// TIA Portal project "Blending_Process" (V16)

(* hardware
DEVICE "S7-1200 station_1"  S7-1200 Station
   slot 0: "Rack_0"  S7-1200 Rack  Rack  V1.0
   slot 1: "PLC_1"  CPU 1214C DC/DC/DC  6ES7 214-1AG40-0XB0  V4.2
DEVICE "HMI_1"  KTP700 Basic PN
   slot 0: "HMI_1"  KTP700 Basic PN  6AV2 123-2GB03-0AX0  16.0.0.0
   slot 1: "HMI_RT_1"  KTP700 Basic PN  6AV2 123-2GB03-0AX0  16.0.0.0
   slot 5: "HMI_1.IE_CP_1"  PROFINET Interface  16.0.0.0
      slot 1: "PROFINET Interface_1"  PROFINET Interface
         slot 1: "Port_1"  Port
*)

// ===== PLC "PLC_1"  CPU 1214C DC/DC/DC =====

VAR_GLOBAL   // PLC tag table "Default tag table"
   "Tag_1" AT %M2.0 : Bool;
   "Tag_2" AT %M2.1 : Bool;
   "RESET_FAULT" AT %M3.3 : Bool;
   "Tag_3" AT %M3.4 : Bool;
   "Reset_Fault_2" AT %M3.5 : Bool;
   "RSET_FAULT_DRAIN" AT %M3.6 : Bool;
   "iq_rMotor_Speed" AT %MD1 : Real;
   "i_xMix_Motor_Stop" AT %I4.0 : Bool;
   "q_xMix_Motor_Stop" AT %Q6.5 : Bool;
   "Tag_4" AT %M50.1 : Bool;
   "Tag_5" AT %M100.0 : Bool;
   "Tag_6" AT %M101.0 : Bool;
   "Tag_7" AT %M102.0 : Bool;
   "Tag_8" AT %M103.0 : Bool;
   "Tag_9" AT %M104.0 : Bool;
   "Tag_10" AT %M110.0 : Bool;
   "Tag_11" AT %M113.0 : Bool;
   "Tag_12" AT %M115.0 : Bool;
   "_iCount_Motor" AT %MW130 : Int;
   "_iCount_Pump1" AT %MW115 : Int;
   "_iCount_Pump2" AT %MW118 : Int;
   "Drain" AT %M74.0 : Bool;
   "Tag_13" AT %M120.0 : Bool;
END_VAR

VAR_GLOBAL   // PLC tag table "Inputs Equipment"
   "i_xSupply_InletValve_Open_A1" AT %I0.1 : Bool;
   "i_xSupply_FeedPump_Running_A1" AT %I2.1 : Bool;
   "i_xSupply_FeedValve_Open_A1" AT %I0.0 : Bool;
   "i_xSupply_FlowSensor_A1" AT %I0.5 : Bool;
   "i_xMix_Motor_Running" AT %I4.1 : Bool;
   "i_xDrain_SolenoidValve_Open" AT %I2.5 : Bool;
   "i_xSupply_InletValve_Open_A2" AT %I0.3 : Bool;
   "i_xSupply_FeedPump_Running_A2" AT %I2.7 : Bool;
   "i_xSupply_FeedValve_Open_A2" AT %I0.2 : Bool;
   "i_xSupply_FlowSensor_A2" AT %I0.6 : Bool;
   "i_xMix_Tank_EmptySensor" AT %I0.4 : Bool;
   "i_rMix_Motor_Voltage" AT %MD10 : Real;
   "i_rMix_Tank_Level" AT %MD64 : Real;
   "i_xSupply_FeedPump_Ready_A1" AT %I3.5 : Bool;
   "i_xSupply_FeedPump_Ready_A2" AT %I3.6 : Bool;
   "i_xDrain_SolenoidValve_Close" AT %I2.3 : Bool;
END_VAR

VAR_GLOBAL   // PLC tag table "Outputs Equipment"
   "q_xSupply_FeedPump_Start_A1" AT %Q3.0 : Bool;
   "q_xMix_Motor_Start" AT %Q6.4 : Bool;
   "q_xDrain_SolenoidValve_Open" AT %Q3.7 : Bool;
   "q_xSupply_FeedPump_Start_A2" AT %Q3.1 : Bool;
   "q_xSupply_InletValve_Open_A2" AT %Q3.3 : Bool;
   "q_xSupply_FeedValve_Open_A2" AT %Q3.5 : Bool;
   "q_xSupply_FeedPump_Stop_A1" AT %Q6.0 : Bool;
   "q_xSupply_FeedPump_Stop_A2" AT %Q6.1 : Bool;
   "q_xDrain_SolenoidValve_Close" AT %Q2.7 : Bool;
   "q_xSupply_FeedValve_Open_A1" AT %Q3.4 : Bool;
   "q_xSupply_InletValve_Open_A1" AT %Q3.2 : Bool;
   "iq_xMix_Tank_FullSensor" AT %I7.7 : Bool;
   "iq_rWater_Level" AT %MD7 : Real;
END_VAR

VAR_GLOBAL   // PLC tag table "Inputs Machine"
   "i_xButtonFeedPump_Start_A1" AT %I30.3 : Bool;
   "i_xButtonFeedPump_Stop_A1" AT %I30.4 : Bool;
   "i_xButtonMotor_Start" AT %I30.0 : Bool;
   "i_xButtonMotor_Stop" AT %I30.1 : Bool;
   "i_xButtonSolenoidValve_Start" AT %I31.0 : Bool;
   "i_xButtonSolenoidValve_Stop" AT %I31.1 : Bool;
   "i_xButtonMaintenanceLamp_Stop" AT %I10.6 : Bool;
   "i_xButton_Emergency" AT %I10.7 : Bool;
   "i_xButtonFeedPump_Start_A2" AT %I30.5 : Bool;
   "i_xButtonFeedPump_Stop_A2" AT %I30.6 : Bool;
   "i_xButton_Reset" AT %I30.2 : Bool;
   "i_xButton_Turn/off_Maintenance_Pump" AT %I31.3 : Bool;
   "i_xButton_Turn/off_Maintenance_Motor" AT %I31.2 : Bool;
   "i_xFull_Sensor" AT %I8.0 : Bool;
END_VAR

VAR_GLOBAL   // PLC tag table "Outputs Machine"
   "q_xLamp_Running" AT %Q4.0 : Bool;
   "q_xLamp_Faulted" AT %Q4.1 : Bool;
   "q_xLamp_Pump_Start_A1" AT %Q4.2 : Bool;
   "q_xLamp_Pump_Stop_A1" AT %Q4.3 : Bool;
   "q_xLamp_Pump_Start_A2" AT %Q4.4 : Bool;
   "q_xLamp_Pump_Stop_A2" AT %Q4.5 : Bool;
   "q_xLamp_Motor_Start" AT %Q4.6 : Bool;
   "q_xLampSolenoidValve_Start" AT %Q5.0 : Bool;
   "q_xLampSolenoidValve_Stop" AT %Q5.1 : Bool;
   "q_xLamp_Pump_Maintain_A1" AT %Q5.2 : Bool;
   "q_xLamp_Pump_Maintain_A2" AT %Q5.3 : Bool;
   "q_xLamp_Motor_Stop" AT %Q4.7 : Bool;
   "q_xLamp_Motor_Maintain" AT %Q5.4 : Bool;
   "q_xLamp_Tank_Full" AT %Q5.5 : Bool;
   "q_xLamp_Tank_Empty" AT %Q5.6 : Bool;
   "q_xLamp_Emergency" AT %Q5.7 : Bool;
   "q_xDisp_Tank_Level" AT %QD60 : Real;
   "q_xDisp_Motor_Speed" AT %QD64 : Real;
   "q_xMaintain_Lamp_Motor" AT %Q10.1 : Bool;
   "q_xMaintain_Lamp_Pump" AT %Q10.2 : Bool;
   "q_xLamp_Fault" AT %Q120.1 : Bool;
END_VAR

// folder: Equipment

TYPE "UDT_Supply"
   STRUCT
      Sts : Struct
         xPumpRunning : Bool;
         xPumpReady : Bool;
         xInletValveOpen : Bool;
         xFeedValveOpen : Bool;
         xFlowSensor : Bool;
         xFauted : Bool;
      END_STRUCT;
      Cmd : Struct
         xSpare : Bool;
         xStart_Pump : Bool;
         xStop_Pump : Bool;
      END_STRUCT;
      Cfg : Struct
         xSpare : Bool;
      END_STRUCT;
      Flt : Struct
         wTrigger : Word;
      END_STRUCT;
   END_STRUCT;
END_TYPE

TYPE "UDT_Mix"
   STRUCT
      Sts : Struct
         xMotorRunning : Bool;
         xMotorReady : Bool;
         iLevel : Int;
         xFullLevel : Bool;
         xEmptyLevel : Bool;
         xFaulted : Bool;
      END_STRUCT;
      Cmd : Struct
         xSpare : Bool;
         xStart_Motor : Bool;
         xStop_Motor : Bool;
      END_STRUCT;
      Cfg : Struct
         xSpare : Bool;
      END_STRUCT;
      Flt : Struct
         wTrigger : Word;
      END_STRUCT;
   END_STRUCT;
END_TYPE

TYPE "UDT_Drain"
   STRUCT
      Sts : Struct
         xSolenoidValveOpen : Bool;
         xSolenoidValveClose : Bool;
         xFaulted : Bool;
      END_STRUCT;
      Cmd : Struct
         xSpare : Bool;
         xStart_SolenoidValve : Bool;
         xStop_SsolenoidValve : Bool;
      END_STRUCT;
      Cfg : Struct
         xSpare : Bool;
      END_STRUCT;
      Flt : Struct
         wTrigger : Word;
      END_STRUCT;
   END_STRUCT;
END_TYPE

// folder: Machine

TYPE "UDT_Statehandler"
   STRUCT
      State : Struct
         xMaintenance_Pump : Bool;
         xMaintenance_Motor : Bool;
         xReady_Pump_A1 : Bool;
         xReady_Pump_A2 : Bool;
         xReady_Motor : Bool;
         xReady_SolenoidValve : Bool;
         xRunning_Pump_A1 : Bool;
         xRunning_Pump_A2 : Bool;
         xRunning_Motor : Bool;
         xRunning_SolenoidValve : Bool;
         xFaulted : Bool;
         xReset : Bool;
      END_STRUCT;
      Cmd : Struct
         xStart : Bool;
         xStop : Bool;
         xReset : Bool;
         xMaintain : Bool;
         xStart_Pump_A1 : Bool;
         xStart_Pump_A2 : Bool;
         xStart_Motor : Bool;
         xStart_SolenoidValve : Bool;
         xStop_Pump_A1 : Bool;
         xStop_Pump_A2 : Bool;
         xStop_Motor : Bool;
         xStop_Solenoid : Bool;
      END_STRUCT;
   END_STRUCT;
END_TYPE

// folder: 00 Machine

DATA_BLOCK "Instance Machine Modules_DB"   // DB3
{ S7_Optimized_Access := 'TRUE' }
VERSION : 0.1
// stored: InstanceOfName FB - Machine Modules
"FB - Machine Modules"
BEGIN
END_DATA_BLOCK

// folder: 01 Equipment

DATA_BLOCK "Instance Equipment Modules"   // DB4
{ S7_Optimized_Access := 'TRUE' }
VERSION : 0.1
// stored: InstanceOfName FB - Equipment Modules
"FB - Equipment Modules"
BEGIN
END_DATA_BLOCK

// folder: 01 Equipment/Functions

DATA_BLOCK "FB - Motor's Speed_DB"   // DB16
{ S7_Optimized_Access := 'TRUE' }
VERSION : 0.1
// stored: InstanceOfName FB - Motor's Speed
"FB - Motor's Speed"
BEGIN
   Power := 0.01;
END_DATA_BLOCK

DATA_BLOCK "FB- Water's Level_DB"   // DB17
{ S7_Optimized_Access := 'TRUE' }
VERSION : 0.1
// stored: InstanceOfName FB- Water's Level
"FB- Water's Level"
BEGIN
   i_rQ := 1.0;
   i_rK := 0.01;
   i_rA := 3.0;
   i_iT := 1;
END_DATA_BLOCK

DATA_BLOCK "FB - Agitator_DB"   // DB19
{ S7_Optimized_Access := 'TRUE' }
VERSION : 0.1
// stored: InstanceOfName FB - Agitator Motor
"FB - Agitator Motor"
BEGIN
END_DATA_BLOCK

// folder: 02 Global Data

DATA_BLOCK "DB  - Machine"   // DB1
{ S7_Optimized_Access := 'FALSE' }
VERSION : 0.1
   VAR
      StateHandler : "UDT_Statehandler";
   END_VAR
BEGIN
END_DATA_BLOCK

DATA_BLOCK "DB -  Equipment"   // DB2
{ S7_Optimized_Access := 'FALSE' }
VERSION : 0.1
   VAR
      Supply_A1 : "UDT_Supply";
      Supply_A2 : "UDT_Supply";
      Mix : "UDT_Mix";
      Drain : "UDT_Drain";
   END_VAR
BEGIN
END_DATA_BLOCK

// folder: System blocks/Program resources

DATA_BLOCK "#stOnDelay_Valve_Open"   // DB5
{ S7_Optimized_Access := 'TRUE' }
AUTHOR : Simatic
FAMILY : IEC
NAME : IEC_TMR
VERSION : 1.0
// stored: InstanceOfName IEC_TIMER
"IEC_TIMER"
BEGIN
END_DATA_BLOCK

DATA_BLOCK "#stOnDelay_Flt_Inlet Valve_2_Open"   // DB6
{ S7_Optimized_Access := 'TRUE' }
AUTHOR : Simatic
FAMILY : IEC
NAME : IEC_TMR
VERSION : 1.0
// stored: InstanceOfName IEC_TIMER
"IEC_TIMER"
BEGIN
END_DATA_BLOCK

DATA_BLOCK "#stOnDelay_Flt_FlowSensor_Report"   // DB7
{ S7_Optimized_Access := 'TRUE' }
AUTHOR : Simatic
FAMILY : IEC
NAME : IEC_TMR
VERSION : 1.0
// stored: InstanceOfName IEC_TIMER
"IEC_TIMER"
BEGIN
END_DATA_BLOCK

DATA_BLOCK "#stOnDelay_Flt_Inlet Valve_Open"   // DB8
{ S7_Optimized_Access := 'TRUE' }
AUTHOR : Simatic
FAMILY : IEC
NAME : IEC_TMR
VERSION : 1.0
// stored: InstanceOfName IEC_TIMER
"IEC_TIMER"
BEGIN
END_DATA_BLOCK

DATA_BLOCK "#stOnDelay_Flt_Feed Valve_Open"   // DB9
{ S7_Optimized_Access := 'TRUE' }
AUTHOR : Simatic
FAMILY : IEC
NAME : IEC_TMR
VERSION : 1.0
// stored: InstanceOfName IEC_TIMER
"IEC_TIMER"
BEGIN
END_DATA_BLOCK

DATA_BLOCK "#stOnDelay_Flt_FlowSensor_2_Report"   // DB10
{ S7_Optimized_Access := 'TRUE' }
AUTHOR : Simatic
FAMILY : IEC
NAME : IEC_TMR
VERSION : 1.0
// stored: InstanceOfName IEC_TIMER
"IEC_TIMER"
BEGIN
END_DATA_BLOCK

DATA_BLOCK "stCTU_Pump_Started"   // DB11
{ S7_Optimized_Access := 'TRUE' }
AUTHOR : Simatic
FAMILY : IEC
NAME : CNTR
VERSION : 1.0
// stored: InstanceOfName IEC_COUNTER
"IEC_COUNTER"
BEGIN
END_DATA_BLOCK

DATA_BLOCK "#stOnDelay_Valve_2_Open"   // DB12
{ S7_Optimized_Access := 'TRUE' }
AUTHOR : Simatic
FAMILY : IEC
NAME : IEC_TMR
VERSION : 1.0
// stored: InstanceOfName IEC_TIMER
"IEC_TIMER"
BEGIN
END_DATA_BLOCK

DATA_BLOCK "#stOnDelay_Flt_Feed Valve_2_Open"   // DB13
{ S7_Optimized_Access := 'TRUE' }
AUTHOR : Simatic
FAMILY : IEC
NAME : IEC_TMR
VERSION : 1.0
// stored: InstanceOfName IEC_TIMER
"IEC_TIMER"
BEGIN
END_DATA_BLOCK

DATA_BLOCK "stCTU_Pump_2_Started"   // DB14
{ S7_Optimized_Access := 'TRUE' }
AUTHOR : Simatic
FAMILY : IEC
NAME : CNTR
VERSION : 1.0
// stored: InstanceOfName IEC_COUNTER
"IEC_COUNTER"
BEGIN
END_DATA_BLOCK

DATA_BLOCK "stOnDelay_Flt_Solenoid_Report"   // DB15
{ S7_Optimized_Access := 'TRUE' }
AUTHOR : Simatic
FAMILY : IEC
NAME : IEC_TMR
VERSION : 1.0
// stored: InstanceOfName IEC_TIMER
"IEC_TIMER"
BEGIN
END_DATA_BLOCK

DATA_BLOCK "20s_Timer_DB"   // DB20
{ S7_Optimized_Access := 'TRUE' }
AUTHOR : Simatic
FAMILY : IEC
NAME : IEC_TMR
VERSION : 1.0
// stored: InstanceOfName IEC_TIMER
"IEC_TIMER"
BEGIN
END_DATA_BLOCK

DATA_BLOCK "stCTU_Motor_Started"   // DB21
{ S7_Optimized_Access := 'TRUE' }
AUTHOR : Simatic
FAMILY : IEC
NAME : CNTR
VERSION : 1.0
// stored: InstanceOfName IEC_COUNTER
"IEC_COUNTER"
BEGIN
END_DATA_BLOCK

// folder: (top level)

ORGANIZATION_BLOCK "Main"   // OB1, LAD, ProgramCycle
TITLE = "Main Program Sweep (Cycle)"
{ S7_Optimized_Access := 'TRUE' }
VERSION : 0.1
   VAR_INPUT
      Initial_Call : Bool;   // Initial call of this OB
      Remanence : Bool;   // =True, if remanent data are available
   END_VAR
BEGIN

REGION Network 1
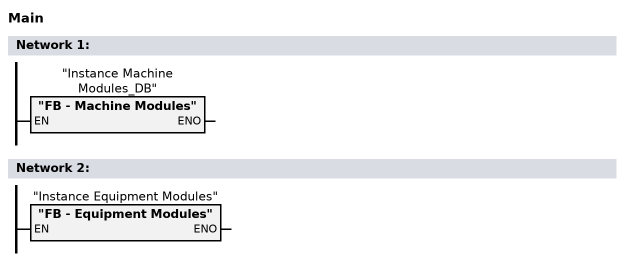
   RUNG wire#powerrail
      "Instance Machine Modules_DB"()
   END_RUNG
   // the same network as SCL:
   "Instance Machine Modules_DB"();   // "FB - Machine Modules"
END_REGION

REGION Network 2
   RUNG wire#powerrail
      "Instance Equipment Modules"()
   END_RUNG
   // the same network as SCL:
   "Instance Equipment Modules"();   // "FB - Equipment Modules"
END_REGION
END_ORGANIZATION_BLOCK

// folder: 00 Machine

FUNCTION_BLOCK "FB - Machine Modules"   // FB1, LAD
{ S7_Optimized_Access := 'TRUE' }
VERSION : 0.1
   VAR
      "Instance StateHandler" : "FB - StateHandler";
      "FB - StateHandler_Instance" : "FB - StateHandler";
      "FB - StateHandler_Instance_1" : "FB - StateHandler";
   END_VAR
BEGIN

REGION Network 1
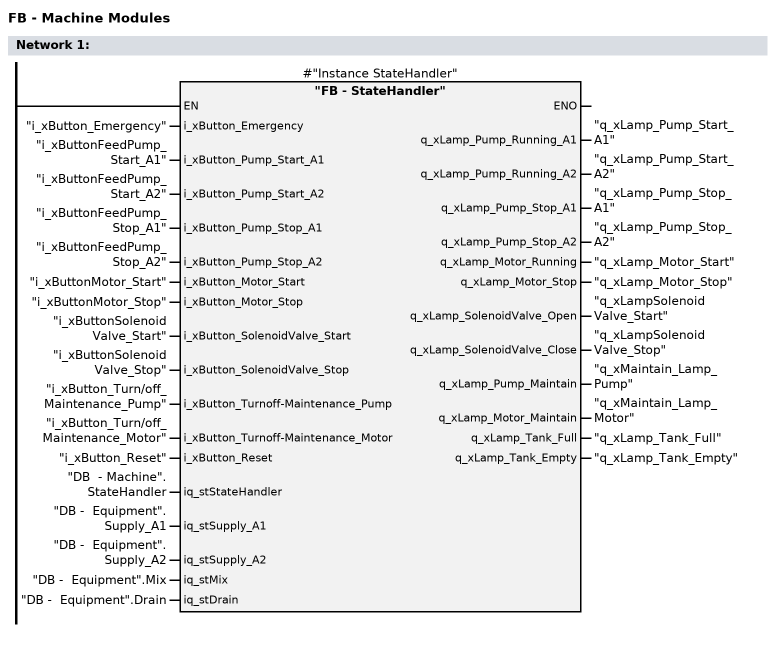
   RUNG wire#powerrail
      #"Instance StateHandler"(i_xButton_Emergency := "i_xButton_Emergency", i_xButton_Pump_Start_A1 := "i_xButtonFeedPump_Start_A1", i_xButton_Pump_Start_A2 := "i_xButtonFeedPump_Start_A2", i_xButton_Pump_Stop_A1 := "i_xButtonFeedPump_Stop_A1", i_xButton_Pump_Stop_A2 := "i_xButtonFeedPump_Stop_A2", i_xButton_Motor_Start := "i_xButtonMotor_Start", i_xButton_Motor_Stop := "i_xButtonMotor_Stop", i_xButton_SolenoidValve_Start := "i_xButtonSolenoidValve_Start", i_xButton_SolenoidValve_Stop := "i_xButtonSolenoidValve_Stop", "i_xButton_Turnoff-Maintenance_Pump" := "i_xButton_Turn/off_Maintenance_Pump", "i_xButton_Turnoff-Maintenance_Motor" := "i_xButton_Turn/off_Maintenance_Motor", i_xButton_Reset := "i_xButton_Reset", iq_stStateHandler := "DB  - Machine".StateHandler, iq_stSupply_A1 := "DB -  Equipment".Supply_A1, iq_stSupply_A2 := "DB -  Equipment".Supply_A2, iq_stMix := "DB -  Equipment".Mix, iq_stDrain := "DB -  Equipment".Drain, q_xLamp_Pump_Running_A1 => "q_xLamp_Pump_Start_A1", q_xLamp_Pump_Running_A2 => "q_xLamp_Pump_Start_A2", q_xLamp_Pump_Stop_A1 => "q_xLamp_Pump_Stop_A1", q_xLamp_Pump_Stop_A2 => "q_xLamp_Pump_Stop_A2", q_xLamp_Motor_Running => "q_xLamp_Motor_Start", q_xLamp_Motor_Stop => "q_xLamp_Motor_Stop", q_xLamp_SolenoidValve_Open => "q_xLampSolenoidValve_Start", q_xLamp_SolenoidValve_Close => "q_xLampSolenoidValve_Stop", q_xLamp_Pump_Maintain => "q_xMaintain_Lamp_Pump", q_xLamp_Motor_Maintain => "q_xMaintain_Lamp_Motor", q_xLamp_Tank_Full => "q_xLamp_Tank_Full", q_xLamp_Tank_Empty => "q_xLamp_Tank_Empty")
   END_RUNG
   // the same network as SCL:
   #"Instance StateHandler"(i_xButton_Emergency := "i_xButton_Emergency",   // "FB - StateHandler"
                           i_xButton_Pump_Start_A1 := "i_xButtonFeedPump_Start_A1",
                           i_xButton_Pump_Start_A2 := "i_xButtonFeedPump_Start_A2",
                           i_xButton_Pump_Stop_A1 := "i_xButtonFeedPump_Stop_A1",
                           i_xButton_Pump_Stop_A2 := "i_xButtonFeedPump_Stop_A2",
                           i_xButton_Motor_Start := "i_xButtonMotor_Start",
                           i_xButton_Motor_Stop := "i_xButtonMotor_Stop",
                           i_xButton_SolenoidValve_Start := "i_xButtonSolenoidValve_Start",
                           i_xButton_SolenoidValve_Stop := "i_xButtonSolenoidValve_Stop",
                           "i_xButton_Turnoff-Maintenance_Pump" := "i_xButton_Turn/off_Maintenance_Pump",
                           "i_xButton_Turnoff-Maintenance_Motor" := "i_xButton_Turn/off_Maintenance_Motor",
                           i_xButton_Reset := "i_xButton_Reset",
                           iq_stStateHandler := "DB  - Machine".StateHandler,
                           iq_stSupply_A1 := "DB -  Equipment".Supply_A1,
                           iq_stSupply_A2 := "DB -  Equipment".Supply_A2,
                           iq_stMix := "DB -  Equipment".Mix,
                           iq_stDrain := "DB -  Equipment".Drain,
                           q_xLamp_Pump_Running_A1 => "q_xLamp_Pump_Start_A1",
                           q_xLamp_Pump_Running_A2 => "q_xLamp_Pump_Start_A2",
                           q_xLamp_Pump_Stop_A1 => "q_xLamp_Pump_Stop_A1",
                           q_xLamp_Pump_Stop_A2 => "q_xLamp_Pump_Stop_A2",
                           q_xLamp_Motor_Running => "q_xLamp_Motor_Start",
                           q_xLamp_Motor_Stop => "q_xLamp_Motor_Stop",
                           q_xLamp_SolenoidValve_Open => "q_xLampSolenoidValve_Start",
                           q_xLamp_SolenoidValve_Close => "q_xLampSolenoidValve_Stop",
                           q_xLamp_Pump_Maintain => "q_xMaintain_Lamp_Pump",
                           q_xLamp_Motor_Maintain => "q_xMaintain_Lamp_Motor",
                           q_xLamp_Tank_Full => "q_xLamp_Tank_Full",
                           q_xLamp_Tank_Empty => "q_xLamp_Tank_Empty");
END_REGION
END_FUNCTION_BLOCK

// folder: 00 Machine/Functions

FUNCTION_BLOCK "FB - StateHandler"   // FB2, LAD
{ S7_Optimized_Access := 'TRUE' }
VERSION : 0.1
   VAR_INPUT
      i_xButton_Emergency : Bool;
      i_xButton_Pump_Start_A1 : Bool;
      i_xButton_Pump_Start_A2 : Bool;
      i_xButton_Pump_Stop_A1 : Bool;
      i_xButton_Pump_Stop_A2 : Bool;
      i_xButton_Motor_Start : Bool;
      i_xButton_Motor_Stop : Bool;
      i_xButton_SolenoidValve_Start : Bool;
      i_xButton_SolenoidValve_Stop : Bool;
      "i_xButton_Turnoff-Maintenance_Pump" : Bool;
      "i_xButton_Turnoff-Maintenance_Motor" : Bool;
      i_xButton_Reset : Bool;
   END_VAR
   VAR_OUTPUT
      q_xLamp_Pump_Running_A1 : Bool;
      q_xLamp_Pump_Running_A2 : Bool;
      q_xLamp_Pump_Stop_A1 : Bool;
      q_xLamp_Pump_Stop_A2 : Bool;
      q_xLamp_Motor_Running : Bool;
      q_xLamp_Motor_Stop : Bool;
      q_xLamp_SolenoidValve_Open : Bool;
      q_xLamp_SolenoidValve_Close : Bool;
      q_xLamp_Pump_Maintain : Bool;
      q_xLamp_Motor_Maintain : Bool;
      q_xLamp_Tank_Full : Bool;
      q_xLamp_Tank_Empty : Bool;
   END_VAR
   VAR_IN_OUT
      iq_stStateHandler : "UDT_Statehandler";
      iq_stSupply_A1 : "UDT_Supply";
      iq_stSupply_A2 : "UDT_Supply";
      iq_stMix : "UDT_Mix";
      iq_stDrain : "UDT_Drain";
   END_VAR
   VAR
      iState_Pump_A1 : Int;
      iState_Pump_A2 : Int;
      iState_Motor : Int;
      iState_SolenoidValve : Int;
      stOnDelay_Reset : TON_TIME;
      stOnDelay_Reset_Motor : TON_TIME;
      stOnDelay_Reset_A1 : TON_TIME;
      stOnDelay_Reset_A2 : TON_TIME;
   END_VAR
BEGIN

REGION Network 1: CONTROL - Start Operation
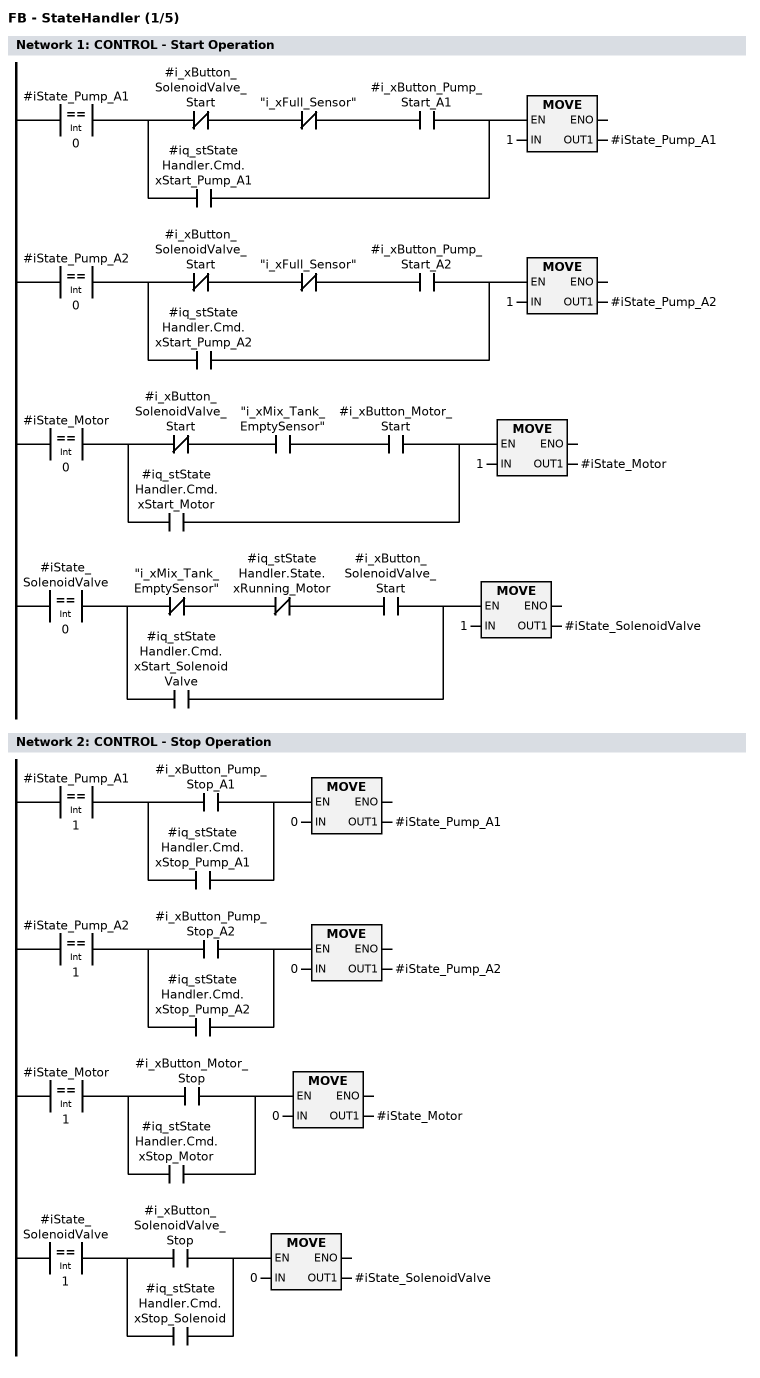
   RUNG wire#powerrail
      { S7_Templates := "SrcType := Int" } EQ_Contact(in1 := #iState_Pump_A1, in2 := 0)
      wire#w1
      I_Contact( #i_xButton_SolenoidValve_Start )
      I_Contact( "i_xFull_Sensor" )
      Contact( #i_xButton_Pump_Start_A1 )
      wire#w2
      Move(in := 1, out1 => #iState_Pump_A1)
   END_RUNG
   RUNG wire#w1
      Contact( #iq_stStateHandler.Cmd.xStart_Pump_A1 )
   END_RUNG wire#w2
   RUNG wire#powerrail
      { S7_Templates := "SrcType := Int" } EQ_Contact(in1 := #iState_Pump_A2, in2 := 0)
      wire#w3
      I_Contact( #i_xButton_SolenoidValve_Start )
      I_Contact( "i_xFull_Sensor" )
      Contact( #i_xButton_Pump_Start_A2 )
      wire#w4
      Move(in := 1, out1 => #iState_Pump_A2)
   END_RUNG
   RUNG wire#w3
      Contact( #iq_stStateHandler.Cmd.xStart_Pump_A2 )
   END_RUNG wire#w4
   RUNG wire#powerrail
      { S7_Templates := "SrcType := Int" } EQ_Contact(in1 := #iState_Motor, in2 := 0)
      wire#w5
      I_Contact( #i_xButton_SolenoidValve_Start )
      Contact( "i_xMix_Tank_EmptySensor" )
      Contact( #i_xButton_Motor_Start )
      wire#w6
      Move(in := 1, out1 => #iState_Motor)
   END_RUNG
   RUNG wire#w5
      Contact( #iq_stStateHandler.Cmd.xStart_Motor )
   END_RUNG wire#w6
   RUNG wire#powerrail
      { S7_Templates := "SrcType := Int" } EQ_Contact(in1 := #iState_SolenoidValve, in2 := 0)
      wire#w7
      I_Contact( "i_xMix_Tank_EmptySensor" )
      I_Contact( #iq_stStateHandler.State.xRunning_Motor )
      Contact( #i_xButton_SolenoidValve_Start )
      wire#w8
      Move(in := 1, out1 => #iState_SolenoidValve)
   END_RUNG
   RUNG wire#w7
      Contact( #iq_stStateHandler.Cmd.xStart_SolenoidValve )
   END_RUNG wire#w8
   // the same network as SCL:
   IF (#iState_Pump_A1 = 0) AND ((NOT #i_xButton_SolenoidValve_Start AND NOT "i_xFull_Sensor" AND #i_xButton_Pump_Start_A1) OR #iq_stStateHandler.Cmd.xStart_Pump_A1) THEN
       #iState_Pump_A1 := 1;
   END_IF;
   IF (#iState_Pump_A2 = 0) AND ((NOT #i_xButton_SolenoidValve_Start AND NOT "i_xFull_Sensor" AND #i_xButton_Pump_Start_A2) OR #iq_stStateHandler.Cmd.xStart_Pump_A2) THEN
       #iState_Pump_A2 := 1;
   END_IF;
   IF (#iState_Motor = 0) AND ((NOT #i_xButton_SolenoidValve_Start AND "i_xMix_Tank_EmptySensor" AND #i_xButton_Motor_Start) OR #iq_stStateHandler.Cmd.xStart_Motor) THEN
       #iState_Motor := 1;
   END_IF;
   IF (#iState_SolenoidValve = 0) AND ((NOT "i_xMix_Tank_EmptySensor" AND NOT #iq_stStateHandler.State.xRunning_Motor AND #i_xButton_SolenoidValve_Start) OR #iq_stStateHandler.Cmd.xStart_SolenoidValve) THEN
       #iState_SolenoidValve := 1;
   END_IF;
END_REGION

REGION Network 2: CONTROL - Stop Operation
   RUNG wire#powerrail
      { S7_Templates := "SrcType := Int" } EQ_Contact(in1 := #iState_Pump_A1, in2 := 1)
      wire#w1
      Contact( #i_xButton_Pump_Stop_A1 )
      wire#w2
      Move(in := 0, out1 => #iState_Pump_A1)
   END_RUNG
   RUNG wire#w1
      Contact( #iq_stStateHandler.Cmd.xStop_Pump_A1 )
   END_RUNG wire#w2
   RUNG wire#powerrail
      { S7_Templates := "SrcType := Int" } EQ_Contact(in1 := #iState_Pump_A2, in2 := 1)
      wire#w3
      Contact( #i_xButton_Pump_Stop_A2 )
      wire#w4
      Move(in := 0, out1 => #iState_Pump_A2)
   END_RUNG
   RUNG wire#w3
      Contact( #iq_stStateHandler.Cmd.xStop_Pump_A2 )
   END_RUNG wire#w4
   RUNG wire#powerrail
      { S7_Templates := "SrcType := Int" } EQ_Contact(in1 := #iState_Motor, in2 := 1)
      wire#w5
      Contact( #i_xButton_Motor_Stop )
      wire#w6
      Move(in := 0, out1 => #iState_Motor)
   END_RUNG
   RUNG wire#w5
      Contact( #iq_stStateHandler.Cmd.xStop_Motor )
   END_RUNG wire#w6
   RUNG wire#powerrail
      { S7_Templates := "SrcType := Int" } EQ_Contact(in1 := #iState_SolenoidValve, in2 := 1)
      wire#w7
      Contact( #i_xButton_SolenoidValve_Stop )
      wire#w8
      Move(in := 0, out1 => #iState_SolenoidValve)
   END_RUNG
   RUNG wire#w7
      Contact( #iq_stStateHandler.Cmd.xStop_Solenoid )
   END_RUNG wire#w8
   // the same network as SCL:
   IF (#iState_Pump_A1 = 1) AND (#i_xButton_Pump_Stop_A1 OR #iq_stStateHandler.Cmd.xStop_Pump_A1) THEN
       #iState_Pump_A1 := 0;
   END_IF;
   IF (#iState_Pump_A2 = 1) AND (#i_xButton_Pump_Stop_A2 OR #iq_stStateHandler.Cmd.xStop_Pump_A2) THEN
       #iState_Pump_A2 := 0;
   END_IF;
   IF (#iState_Motor = 1) AND (#i_xButton_Motor_Stop OR #iq_stStateHandler.Cmd.xStop_Motor) THEN
       #iState_Motor := 0;
   END_IF;
   IF (#iState_SolenoidValve = 1) AND (#i_xButton_SolenoidValve_Stop OR #iq_stStateHandler.Cmd.xStop_Solenoid) THEN
       #iState_SolenoidValve := 0;
   END_IF;
END_REGION

REGION Network 3: CONTROL - Application Faulted
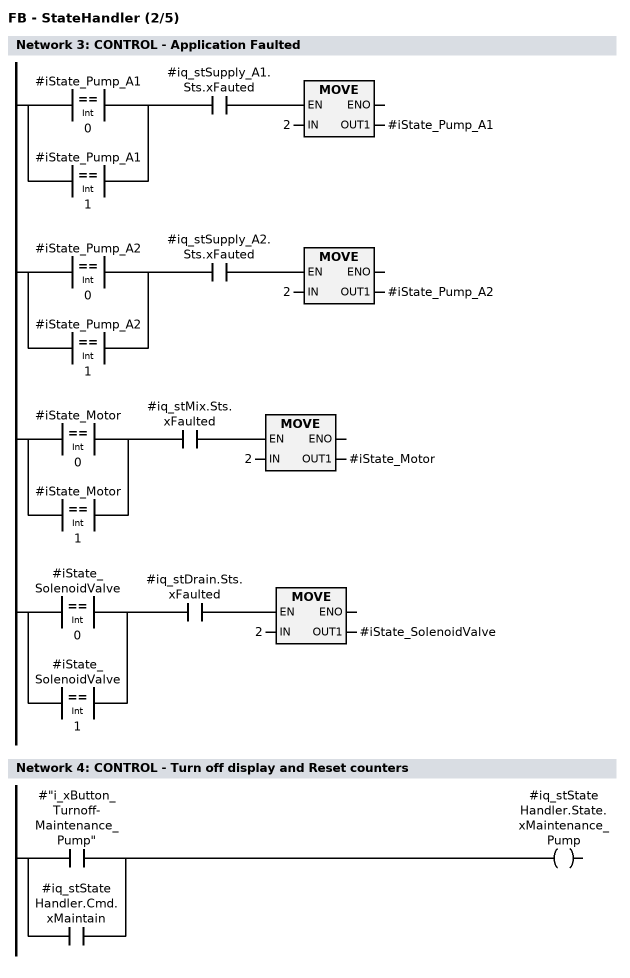
   RUNG wire#powerrail
      { S7_Templates := "SrcType := Int" } EQ_Contact(in1 := #iState_Pump_A1, in2 := 0)
      wire#w1
      Contact( #iq_stSupply_A1.Sts.xFauted )
      Move(in := 2, out1 => #iState_Pump_A1)
   END_RUNG
   RUNG wire#powerrail
      { S7_Templates := "SrcType := Int" } EQ_Contact(in1 := #iState_Pump_A1, in2 := 1)
   END_RUNG wire#w1
   RUNG wire#powerrail
      { S7_Templates := "SrcType := Int" } EQ_Contact(in1 := #iState_Pump_A2, in2 := 0)
      wire#w2
      Contact( #iq_stSupply_A2.Sts.xFauted )
      Move(in := 2, out1 => #iState_Pump_A2)
   END_RUNG
   RUNG wire#powerrail
      { S7_Templates := "SrcType := Int" } EQ_Contact(in1 := #iState_Pump_A2, in2 := 1)
   END_RUNG wire#w2
   RUNG wire#powerrail
      { S7_Templates := "SrcType := Int" } EQ_Contact(in1 := #iState_Motor, in2 := 0)
      wire#w3
      Contact( #iq_stMix.Sts.xFaulted )
      Move(in := 2, out1 => #iState_Motor)
   END_RUNG
   RUNG wire#powerrail
      { S7_Templates := "SrcType := Int" } EQ_Contact(in1 := #iState_Motor, in2 := 1)
   END_RUNG wire#w3
   RUNG wire#powerrail
      { S7_Templates := "SrcType := Int" } EQ_Contact(in1 := #iState_SolenoidValve, in2 := 0)
      wire#w4
      Contact( #iq_stDrain.Sts.xFaulted )
      Move(in := 2, out1 => #iState_SolenoidValve)
   END_RUNG
   RUNG wire#powerrail
      { S7_Templates := "SrcType := Int" } EQ_Contact(in1 := #iState_SolenoidValve, in2 := 1)
   END_RUNG wire#w4
   // the same network as SCL:
   IF ((#iState_Pump_A1 = 0) OR (#iState_Pump_A1 = 1)) AND #iq_stSupply_A1.Sts.xFauted THEN
       #iState_Pump_A1 := 2;
   END_IF;
   IF ((#iState_Pump_A2 = 0) OR (#iState_Pump_A2 = 1)) AND #iq_stSupply_A2.Sts.xFauted THEN
       #iState_Pump_A2 := 2;
   END_IF;
   IF ((#iState_Motor = 0) OR (#iState_Motor = 1)) AND #iq_stMix.Sts.xFaulted THEN
       #iState_Motor := 2;
   END_IF;
   IF ((#iState_SolenoidValve = 0) OR (#iState_SolenoidValve = 1)) AND #iq_stDrain.Sts.xFaulted THEN
       #iState_SolenoidValve := 2;
   END_IF;
END_REGION

REGION Network 4: CONTROL - Turn off display and Reset counters
   RUNG wire#powerrail
      Contact( #"i_xButton_Turnoff-Maintenance_Pump" )
      wire#w1
      Coil( #iq_stStateHandler.State.xMaintenance_Pump )
   END_RUNG
   RUNG wire#powerrail
      Contact( #iq_stStateHandler.Cmd.xMaintain )
   END_RUNG wire#w1
   // the same network as SCL:
   #iq_stStateHandler.State.xMaintenance_Pump := #"i_xButton_Turnoff-Maintenance_Pump" OR #iq_stStateHandler.Cmd.xMaintain;
END_REGION

REGION Network 5: STATUS - State Ready
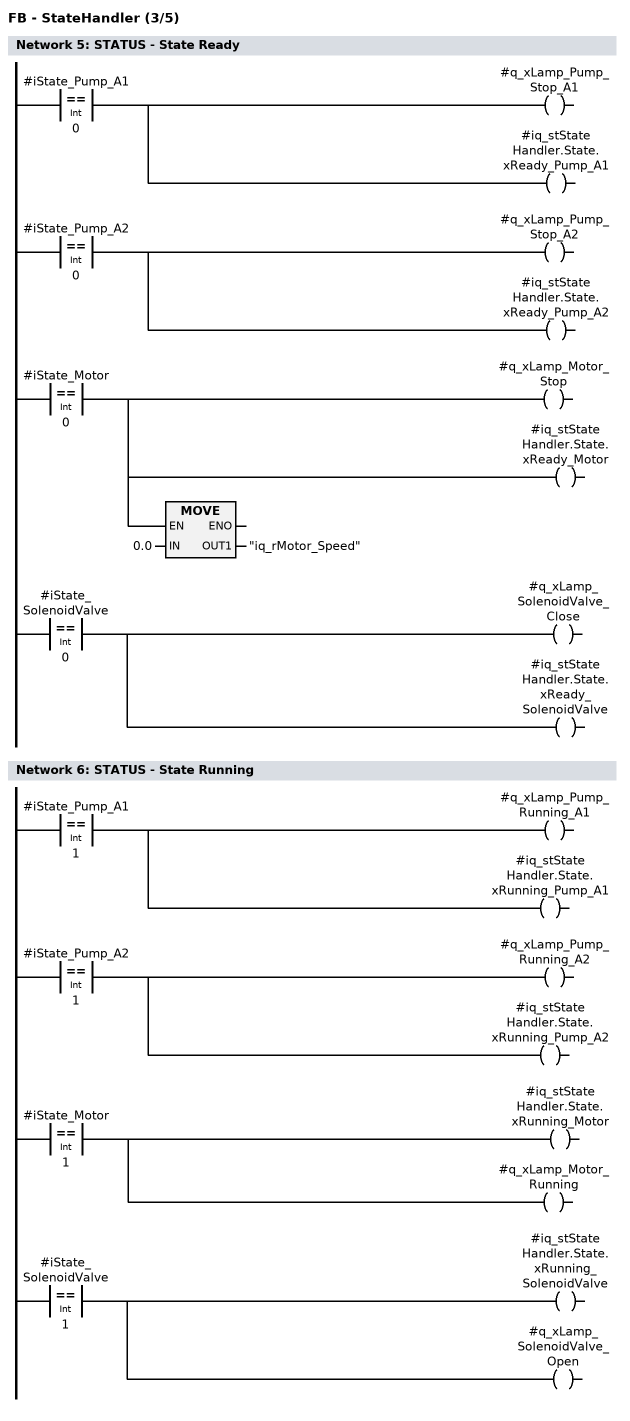
   RUNG wire#powerrail
      { S7_Templates := "SrcType := Int" } EQ_Contact(in1 := #iState_Pump_A1, in2 := 0)
      wire#w1
      Coil( #q_xLamp_Pump_Stop_A1 )
   END_RUNG
   RUNG wire#w1
      Coil( #iq_stStateHandler.State.xReady_Pump_A1 )
   END_RUNG
   RUNG wire#powerrail
      { S7_Templates := "SrcType := Int" } EQ_Contact(in1 := #iState_Pump_A2, in2 := 0)
      wire#w2
      Coil( #q_xLamp_Pump_Stop_A2 )
   END_RUNG
   RUNG wire#w2
      Coil( #iq_stStateHandler.State.xReady_Pump_A2 )
   END_RUNG
   RUNG wire#powerrail
      { S7_Templates := "SrcType := Int" } EQ_Contact(in1 := #iState_Motor, in2 := 0)
      wire#w3
      Coil( #q_xLamp_Motor_Stop )
   END_RUNG
   RUNG wire#w3
      Coil( #iq_stStateHandler.State.xReady_Motor )
   END_RUNG
   RUNG wire#w3
      Move(in := 0.0, out1 => "iq_rMotor_Speed")
   END_RUNG
   RUNG wire#powerrail
      { S7_Templates := "SrcType := Int" } EQ_Contact(in1 := #iState_SolenoidValve, in2 := 0)
      wire#w4
      Coil( #q_xLamp_SolenoidValve_Close )
   END_RUNG
   RUNG wire#w4
      Coil( #iq_stStateHandler.State.xReady_SolenoidValve )
   END_RUNG
   // the same network as SCL:
   #q_xLamp_Pump_Stop_A1 := #iState_Pump_A1 = 0;
   #iq_stStateHandler.State.xReady_Pump_A1 := #q_xLamp_Pump_Stop_A1;
   #q_xLamp_Pump_Stop_A2 := #iState_Pump_A2 = 0;
   #iq_stStateHandler.State.xReady_Pump_A2 := #q_xLamp_Pump_Stop_A2;
   #q_xLamp_Motor_Stop := #iState_Motor = 0;
   #iq_stStateHandler.State.xReady_Motor := #q_xLamp_Motor_Stop;
   IF #q_xLamp_Motor_Stop THEN "iq_rMotor_Speed" := 0.0; END_IF;
   #q_xLamp_SolenoidValve_Close := #iState_SolenoidValve = 0;
   #iq_stStateHandler.State.xReady_SolenoidValve := #q_xLamp_SolenoidValve_Close;
END_REGION

REGION Network 6: STATUS - State Running
   RUNG wire#powerrail
      { S7_Templates := "SrcType := Int" } EQ_Contact(in1 := #iState_Pump_A1, in2 := 1)
      wire#w1
      Coil( #q_xLamp_Pump_Running_A1 )
   END_RUNG
   RUNG wire#w1
      Coil( #iq_stStateHandler.State.xRunning_Pump_A1 )
   END_RUNG
   RUNG wire#powerrail
      { S7_Templates := "SrcType := Int" } EQ_Contact(in1 := #iState_Pump_A2, in2 := 1)
      wire#w2
      Coil( #q_xLamp_Pump_Running_A2 )
   END_RUNG
   RUNG wire#w2
      Coil( #iq_stStateHandler.State.xRunning_Pump_A2 )
   END_RUNG
   RUNG wire#powerrail
      { S7_Templates := "SrcType := Int" } EQ_Contact(in1 := #iState_Motor, in2 := 1)
      wire#w3
      Coil( #iq_stStateHandler.State.xRunning_Motor )
   END_RUNG
   RUNG wire#w3
      Coil( #q_xLamp_Motor_Running )
   END_RUNG
   RUNG wire#powerrail
      { S7_Templates := "SrcType := Int" } EQ_Contact(in1 := #iState_SolenoidValve, in2 := 1)
      wire#w4
      Coil( #iq_stStateHandler.State.xRunning_SolenoidValve )
   END_RUNG
   RUNG wire#w4
      Coil( #q_xLamp_SolenoidValve_Open )
   END_RUNG
   // the same network as SCL:
   #q_xLamp_Pump_Running_A1 := #iState_Pump_A1 = 1;
   #iq_stStateHandler.State.xRunning_Pump_A1 := #q_xLamp_Pump_Running_A1;
   #q_xLamp_Pump_Running_A2 := #iState_Pump_A2 = 1;
   #iq_stStateHandler.State.xRunning_Pump_A2 := #q_xLamp_Pump_Running_A2;
   #iq_stStateHandler.State.xRunning_Motor := #iState_Motor = 1;
   #q_xLamp_Motor_Running := #iq_stStateHandler.State.xRunning_Motor;
   #iq_stStateHandler.State.xRunning_SolenoidValve := #iState_SolenoidValve = 1;
   #q_xLamp_SolenoidValve_Open := #iq_stStateHandler.State.xRunning_SolenoidValve;
END_REGION

REGION Network 7: CONTROL - Reset Request
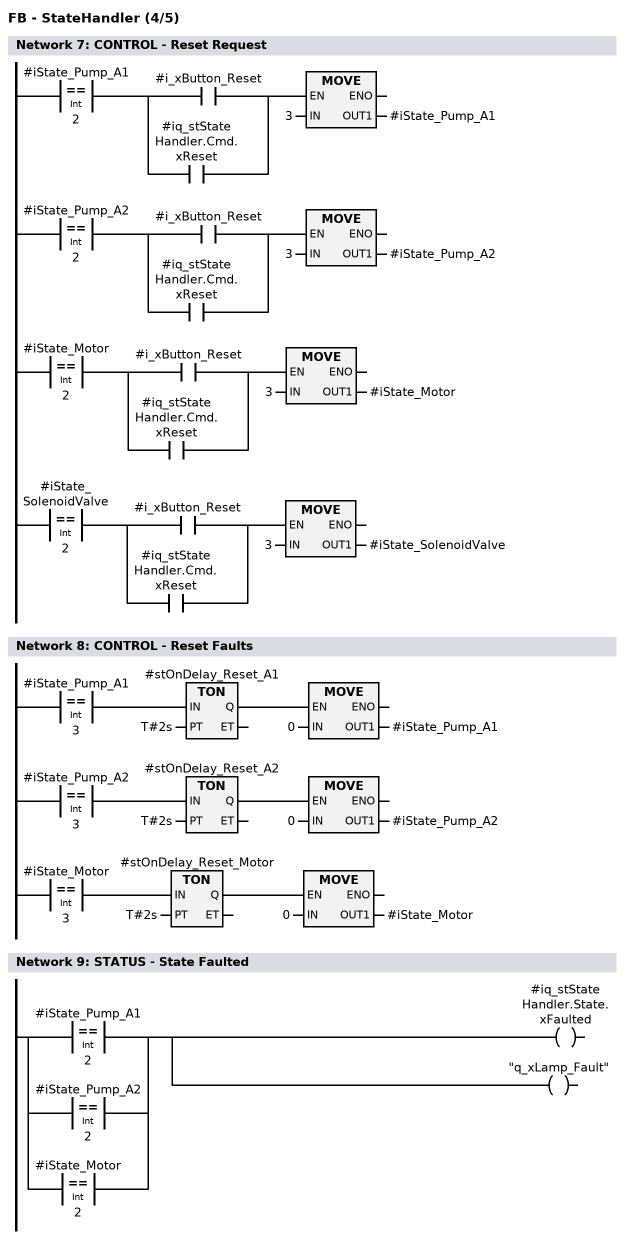
   RUNG wire#powerrail
      { S7_Templates := "SrcType := Int" } EQ_Contact(in1 := #iState_Pump_A1, in2 := 2)
      wire#w1
      Contact( #i_xButton_Reset )
      wire#w2
      Move(in := 3, out1 => #iState_Pump_A1)
   END_RUNG
   RUNG wire#w1
      Contact( #iq_stStateHandler.Cmd.xReset )
   END_RUNG wire#w2
   RUNG wire#powerrail
      { S7_Templates := "SrcType := Int" } EQ_Contact(in1 := #iState_Pump_A2, in2 := 2)
      wire#w3
      Contact( #i_xButton_Reset )
      wire#w4
      Move(in := 3, out1 => #iState_Pump_A2)
   END_RUNG
   RUNG wire#w3
      Contact( #iq_stStateHandler.Cmd.xReset )
   END_RUNG wire#w4
   RUNG wire#powerrail
      { S7_Templates := "SrcType := Int" } EQ_Contact(in1 := #iState_Motor, in2 := 2)
      wire#w5
      Contact( #i_xButton_Reset )
      wire#w6
      Move(in := 3, out1 => #iState_Motor)
   END_RUNG
   RUNG wire#w5
      Contact( #iq_stStateHandler.Cmd.xReset )
   END_RUNG wire#w6
   RUNG wire#powerrail
      { S7_Templates := "SrcType := Int" } EQ_Contact(in1 := #iState_SolenoidValve, in2 := 2)
      wire#w7
      Contact( #i_xButton_Reset )
      wire#w8
      Move(in := 3, out1 => #iState_SolenoidValve)
   END_RUNG
   RUNG wire#w7
      Contact( #iq_stStateHandler.Cmd.xReset )
   END_RUNG wire#w8
   // the same network as SCL:
   IF (#iState_Pump_A1 = 2) AND (#i_xButton_Reset OR #iq_stStateHandler.Cmd.xReset) THEN
       #iState_Pump_A1 := 3;
   END_IF;
   IF (#iState_Pump_A2 = 2) AND (#i_xButton_Reset OR #iq_stStateHandler.Cmd.xReset) THEN
       #iState_Pump_A2 := 3;
   END_IF;
   IF (#iState_Motor = 2) AND (#i_xButton_Reset OR #iq_stStateHandler.Cmd.xReset) THEN
       #iState_Motor := 3;
   END_IF;
   IF (#iState_SolenoidValve = 2) AND (#i_xButton_Reset OR #iq_stStateHandler.Cmd.xReset) THEN
       #iState_SolenoidValve := 3;
   END_IF;
END_REGION

REGION Network 8: CONTROL - Reset Faults
   #stOnDelay_Reset_A1(IN := #iState_Pump_A1 = 3, PT := T#2s);   // TON
   IF #stOnDelay_Reset_A1.Q THEN #iState_Pump_A1 := 0; END_IF;
   #stOnDelay_Reset_A2(IN := #iState_Pump_A2 = 3, PT := T#2s);   // TON
   IF #stOnDelay_Reset_A2.Q THEN #iState_Pump_A2 := 0; END_IF;
   #stOnDelay_Reset_Motor(IN := #iState_Motor = 3, PT := T#2s);   // TON
   IF #stOnDelay_Reset_Motor.Q THEN #iState_Motor := 0; END_IF;
END_REGION

REGION Network 9: STATUS - State Faulted
   RUNG wire#powerrail
      { S7_Templates := "SrcType := Int" } EQ_Contact(in1 := #iState_Pump_A1, in2 := 2)
      wire#w1
      Coil( #iq_stStateHandler.State.xFaulted )
   END_RUNG
   RUNG wire#powerrail
      { S7_Templates := "SrcType := Int" } EQ_Contact(in1 := #iState_Pump_A2, in2 := 2)
   END_RUNG wire#w1
   RUNG wire#powerrail
      { S7_Templates := "SrcType := Int" } EQ_Contact(in1 := #iState_Motor, in2 := 2)
   END_RUNG wire#w1
   RUNG wire#w1
      Coil( "q_xLamp_Fault" )
   END_RUNG
   // the same network as SCL:
   #iq_stStateHandler.State.xFaulted := (#iState_Pump_A1 = 2) OR (#iState_Pump_A2 = 2) OR (#iState_Motor = 2);
   "q_xLamp_Fault" := #iq_stStateHandler.State.xFaulted;
END_REGION

REGION Network 10: STATUS - State Reset
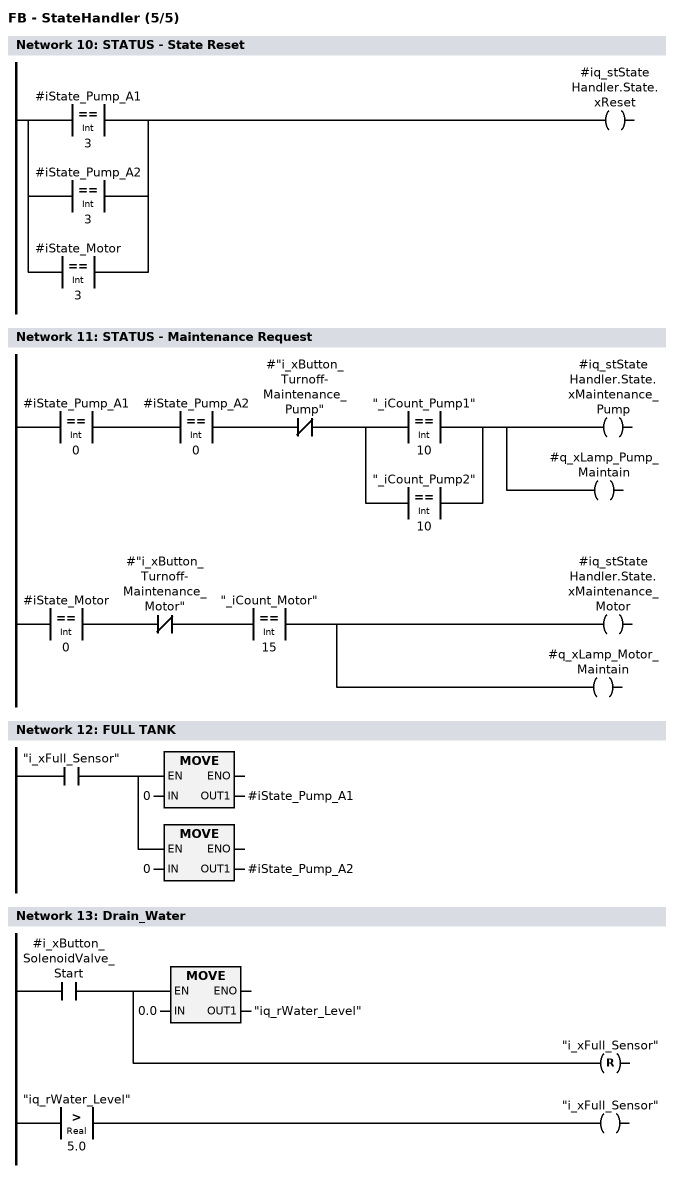
   RUNG wire#powerrail
      { S7_Templates := "SrcType := Int" } EQ_Contact(in1 := #iState_Pump_A1, in2 := 3)
      wire#w1
      Coil( #iq_stStateHandler.State.xReset )
   END_RUNG
   RUNG wire#powerrail
      { S7_Templates := "SrcType := Int" } EQ_Contact(in1 := #iState_Pump_A2, in2 := 3)
   END_RUNG wire#w1
   RUNG wire#powerrail
      { S7_Templates := "SrcType := Int" } EQ_Contact(in1 := #iState_Motor, in2 := 3)
   END_RUNG wire#w1
   // the same network as SCL:
   #iq_stStateHandler.State.xReset := (#iState_Pump_A1 = 3) OR (#iState_Pump_A2 = 3) OR (#iState_Motor = 3);
END_REGION

REGION Network 11: STATUS - Maintenance Request
   RUNG wire#powerrail
      { S7_Templates := "SrcType := Int" } EQ_Contact(in1 := #iState_Pump_A1, in2 := 0)
      { S7_Templates := "SrcType := Int" } EQ_Contact(in1 := #iState_Pump_A2, in2 := 0)
      I_Contact( #"i_xButton_Turnoff-Maintenance_Pump" )
      wire#w1
      { S7_Templates := "SrcType := Int" } EQ_Contact(in1 := "_iCount_Pump1", in2 := 10)
      wire#w2
      Coil( #iq_stStateHandler.State.xMaintenance_Pump )
   END_RUNG
   RUNG wire#w1
      { S7_Templates := "SrcType := Int" } EQ_Contact(in1 := "_iCount_Pump2", in2 := 10)
   END_RUNG wire#w2
   RUNG wire#w2
      Coil( #q_xLamp_Pump_Maintain )
   END_RUNG
   RUNG wire#powerrail
      { S7_Templates := "SrcType := Int" } EQ_Contact(in1 := #iState_Motor, in2 := 0)
      I_Contact( #"i_xButton_Turnoff-Maintenance_Motor" )
      { S7_Templates := "SrcType := Int" } EQ_Contact(in1 := "_iCount_Motor", in2 := 15)
      wire#w3
      Coil( #iq_stStateHandler.State.xMaintenance_Motor )
   END_RUNG
   RUNG wire#w3
      Coil( #q_xLamp_Motor_Maintain )
   END_RUNG
   // the same network as SCL:
   #iq_stStateHandler.State.xMaintenance_Pump := (#iState_Pump_A1 = 0) AND (#iState_Pump_A2 = 0) AND NOT #"i_xButton_Turnoff-Maintenance_Pump" AND (("_iCount_Pump1" = 10) OR ("_iCount_Pump2" = 10));
   #q_xLamp_Pump_Maintain := #iq_stStateHandler.State.xMaintenance_Pump;
   #iq_stStateHandler.State.xMaintenance_Motor := (#iState_Motor = 0) AND NOT #"i_xButton_Turnoff-Maintenance_Motor" AND ("_iCount_Motor" = 15);
   #q_xLamp_Motor_Maintain := #iq_stStateHandler.State.xMaintenance_Motor;
END_REGION

REGION Network 12: FULL TANK
   RUNG wire#powerrail
      Contact( "i_xFull_Sensor" )
      wire#w1
      Move(in := 0, out1 => #iState_Pump_A1)
   END_RUNG
   RUNG wire#w1
      Move(in := 0, out1 => #iState_Pump_A2)
   END_RUNG
   // the same network as SCL:
   IF "i_xFull_Sensor" THEN
       #iState_Pump_A1 := 0;
       #iState_Pump_A2 := 0;
   END_IF;
END_REGION

REGION Network 13: Drain_Water
   RUNG wire#powerrail
      Contact( #i_xButton_SolenoidValve_Start )
      wire#w1
      Move(in := 0.0, out1 => "iq_rWater_Level")
   END_RUNG
   RUNG wire#w1
      R_Coil( "i_xFull_Sensor" )
   END_RUNG
   RUNG wire#powerrail
      { S7_Templates := "SrcType := Real" } GT_Contact(in1 := "iq_rWater_Level", in2 := 5.0)
      Coil( "i_xFull_Sensor" )
   END_RUNG
   // the same network as SCL:
   IF #i_xButton_SolenoidValve_Start THEN
       "iq_rWater_Level" := 0.0;
       "i_xFull_Sensor" := FALSE;
   END_IF;
   "i_xFull_Sensor" := "iq_rWater_Level" > 5.0;
END_REGION
END_FUNCTION_BLOCK

// folder: 01 Equipment

FUNCTION_BLOCK "FB - Equipment Modules"   // FB3, LAD
{ S7_Optimized_Access := 'TRUE' }
VERSION : 0.1
   VAR
      Instance_Supply_A1_Instance : "FB - Supply_A1";
      Instance_Supply_A1 : "FB - Supply_A1";
      Instance_Supply_A2 : "FB - Supply_A2";
      Instance_Drain : "FB - Drain Valve";
   END_VAR
   VAR_TEMP   // added for the SCL form of the ladder/FBD networks
      _w1 : Bool;
      _w2 : Bool;
   END_VAR
BEGIN

REGION Network 1: Supply A1
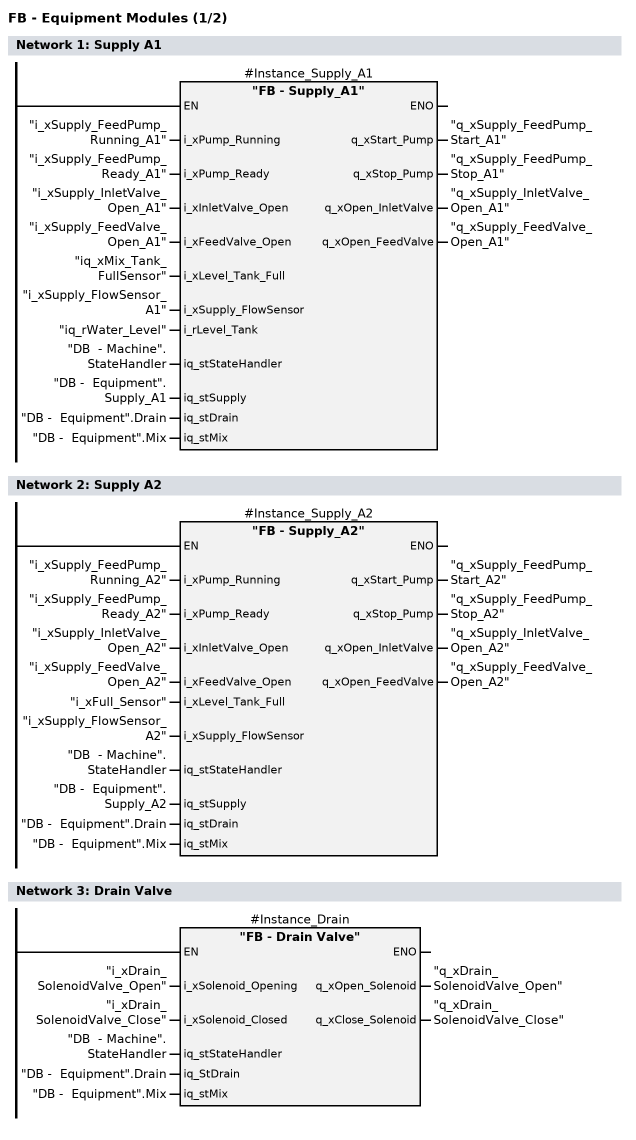
   RUNG wire#powerrail
      #Instance_Supply_A1(i_xPump_Running := "i_xSupply_FeedPump_Running_A1", i_xPump_Ready := "i_xSupply_FeedPump_Ready_A1", i_xInletValve_Open := "i_xSupply_InletValve_Open_A1", i_xFeedValve_Open := "i_xSupply_FeedValve_Open_A1", i_xLevel_Tank_Full := "iq_xMix_Tank_FullSensor", i_xSupply_FlowSensor := "i_xSupply_FlowSensor_A1", i_rLevel_Tank := "iq_rWater_Level", iq_stStateHandler := "DB  - Machine".StateHandler, iq_stSupply := "DB -  Equipment".Supply_A1, iq_stDrain := "DB -  Equipment".Drain, iq_stMix := "DB -  Equipment".Mix, q_xStart_Pump => "q_xSupply_FeedPump_Start_A1", q_xStop_Pump => "q_xSupply_FeedPump_Stop_A1", q_xOpen_InletValve => "q_xSupply_InletValve_Open_A1", q_xOpen_FeedValve => "q_xSupply_FeedValve_Open_A1")
   END_RUNG
   // the same network as SCL:
   #Instance_Supply_A1(i_xPump_Running := "i_xSupply_FeedPump_Running_A1",   // "FB - Supply_A1"
                       i_xPump_Ready := "i_xSupply_FeedPump_Ready_A1",
                       i_xInletValve_Open := "i_xSupply_InletValve_Open_A1",
                       i_xFeedValve_Open := "i_xSupply_FeedValve_Open_A1",
                       i_xLevel_Tank_Full := "iq_xMix_Tank_FullSensor",
                       i_xSupply_FlowSensor := "i_xSupply_FlowSensor_A1",
                       i_rLevel_Tank := "iq_rWater_Level",
                       iq_stStateHandler := "DB  - Machine".StateHandler,
                       iq_stSupply := "DB -  Equipment".Supply_A1,
                       iq_stDrain := "DB -  Equipment".Drain,
                       iq_stMix := "DB -  Equipment".Mix,
                       q_xStart_Pump => "q_xSupply_FeedPump_Start_A1",
                       q_xStop_Pump => "q_xSupply_FeedPump_Stop_A1",
                       q_xOpen_InletValve => "q_xSupply_InletValve_Open_A1",
                       q_xOpen_FeedValve => "q_xSupply_FeedValve_Open_A1");
END_REGION

REGION Network 2: Supply A2
   RUNG wire#powerrail
      #Instance_Supply_A2(i_xPump_Running := "i_xSupply_FeedPump_Running_A2", i_xPump_Ready := "i_xSupply_FeedPump_Ready_A2", i_xInletValve_Open := "i_xSupply_InletValve_Open_A2", i_xFeedValve_Open := "i_xSupply_FeedValve_Open_A2", i_xLevel_Tank_Full := "i_xFull_Sensor", i_xSupply_FlowSensor := "i_xSupply_FlowSensor_A2", iq_stStateHandler := "DB  - Machine".StateHandler, iq_stSupply := "DB -  Equipment".Supply_A2, iq_stDrain := "DB -  Equipment".Drain, iq_stMix := "DB -  Equipment".Mix, q_xStart_Pump => "q_xSupply_FeedPump_Start_A2", q_xStop_Pump => "q_xSupply_FeedPump_Stop_A2", q_xOpen_InletValve => "q_xSupply_InletValve_Open_A2", q_xOpen_FeedValve => "q_xSupply_FeedValve_Open_A2")
   END_RUNG
   // the same network as SCL:
   #Instance_Supply_A2(i_xPump_Running := "i_xSupply_FeedPump_Running_A2",   // "FB - Supply_A2"
                       i_xPump_Ready := "i_xSupply_FeedPump_Ready_A2",
                       i_xInletValve_Open := "i_xSupply_InletValve_Open_A2",
                       i_xFeedValve_Open := "i_xSupply_FeedValve_Open_A2",
                       i_xLevel_Tank_Full := "i_xFull_Sensor",
                       i_xSupply_FlowSensor := "i_xSupply_FlowSensor_A2",
                       iq_stStateHandler := "DB  - Machine".StateHandler,
                       iq_stSupply := "DB -  Equipment".Supply_A2,
                       iq_stDrain := "DB -  Equipment".Drain,
                       iq_stMix := "DB -  Equipment".Mix,
                       q_xStart_Pump => "q_xSupply_FeedPump_Start_A2",
                       q_xStop_Pump => "q_xSupply_FeedPump_Stop_A2",
                       q_xOpen_InletValve => "q_xSupply_InletValve_Open_A2",
                       q_xOpen_FeedValve => "q_xSupply_FeedValve_Open_A2");
END_REGION

REGION Network 3: Drain Valve
   RUNG wire#powerrail
      #Instance_Drain(i_xSolenoid_Opening := "i_xDrain_SolenoidValve_Open", i_xSolenoid_Closed := "i_xDrain_SolenoidValve_Close", iq_stStateHandler := "DB  - Machine".StateHandler, iq_StDrain := "DB -  Equipment".Drain, iq_stMix := "DB -  Equipment".Mix, q_xOpen_Solenoid => "q_xDrain_SolenoidValve_Open", q_xClose_Solenoid => "q_xDrain_SolenoidValve_Close")
   END_RUNG
   // the same network as SCL:
   #Instance_Drain(i_xSolenoid_Opening := "i_xDrain_SolenoidValve_Open",   // "FB - Drain Valve"
                   i_xSolenoid_Closed := "i_xDrain_SolenoidValve_Close",
                   iq_stStateHandler := "DB  - Machine".StateHandler,
                   iq_StDrain := "DB -  Equipment".Drain,
                   iq_stMix := "DB -  Equipment".Mix,
                   q_xOpen_Solenoid => "q_xDrain_SolenoidValve_Open",
                   q_xClose_Solenoid => "q_xDrain_SolenoidValve_Close");
END_REGION

REGION Network 4: Agitator Motor
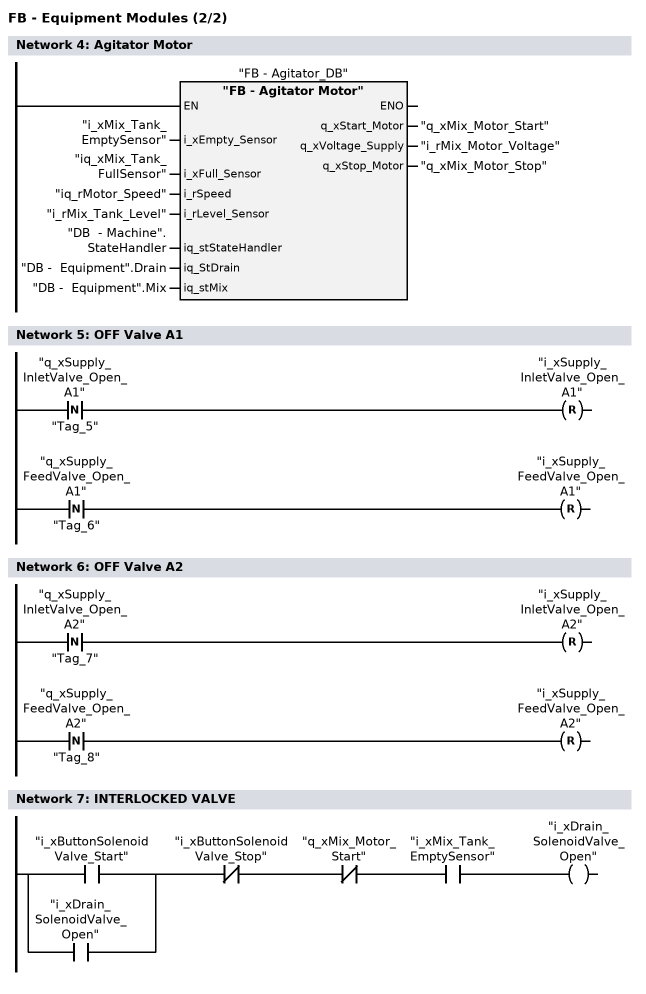
   RUNG wire#powerrail
      "FB - Agitator_DB"(i_xEmpty_Sensor := "i_xMix_Tank_EmptySensor", i_xFull_Sensor := "iq_xMix_Tank_FullSensor", i_rSpeed := "iq_rMotor_Speed", i_rLevel_Sensor := "i_rMix_Tank_Level", iq_stStateHandler := "DB  - Machine".StateHandler, iq_StDrain := "DB -  Equipment".Drain, iq_stMix := "DB -  Equipment".Mix, q_xStart_Motor => "q_xMix_Motor_Start", q_xVoltage_Supply => "i_rMix_Motor_Voltage", q_xStop_Motor => "q_xMix_Motor_Stop")
   END_RUNG
   // the same network as SCL:
   "FB - Agitator_DB"(i_xEmpty_Sensor := "i_xMix_Tank_EmptySensor",   // "FB - Agitator Motor"
                      i_xFull_Sensor := "iq_xMix_Tank_FullSensor",
                      i_rSpeed := "iq_rMotor_Speed",
                      i_rLevel_Sensor := "i_rMix_Tank_Level",
                      iq_stStateHandler := "DB  - Machine".StateHandler,
                      iq_StDrain := "DB -  Equipment".Drain,
                      iq_stMix := "DB -  Equipment".Mix,
                      q_xStart_Motor => "q_xMix_Motor_Start",
                      q_xVoltage_Supply => "i_rMix_Motor_Voltage",
                      q_xStop_Motor => "q_xMix_Motor_Stop");
END_REGION

REGION Network 5: OFF Valve A1
   RUNG wire#powerrail
      N_Contact(operand := "q_xSupply_InletValve_Open_A1", bit := "Tag_5")
      R_Coil( "i_xSupply_InletValve_Open_A1" )
   END_RUNG
   RUNG wire#powerrail
      N_Contact(operand := "q_xSupply_FeedValve_Open_A1", bit := "Tag_6")
      R_Coil( "i_xSupply_FeedValve_Open_A1" )
   END_RUNG
   // the same network as SCL:
   #_w1 := NOT "q_xSupply_InletValve_Open_A1" AND "Tag_5";   // falling edge of "q_xSupply_InletValve_Open_A1"
   "Tag_5" := "q_xSupply_InletValve_Open_A1";
   IF #_w1 THEN "i_xSupply_InletValve_Open_A1" := FALSE; END_IF;
   #_w2 := NOT "q_xSupply_FeedValve_Open_A1" AND "Tag_6";   // falling edge of "q_xSupply_FeedValve_Open_A1"
   "Tag_6" := "q_xSupply_FeedValve_Open_A1";
   IF #_w2 THEN "i_xSupply_FeedValve_Open_A1" := FALSE; END_IF;
END_REGION

REGION Network 6: OFF Valve A2
   RUNG wire#powerrail
      N_Contact(operand := "q_xSupply_InletValve_Open_A2", bit := "Tag_7")
      R_Coil( "i_xSupply_InletValve_Open_A2" )
   END_RUNG
   RUNG wire#powerrail
      N_Contact(operand := "q_xSupply_FeedValve_Open_A2", bit := "Tag_8")
      R_Coil( "i_xSupply_FeedValve_Open_A2" )
   END_RUNG
   // the same network as SCL:
   #_w1 := NOT "q_xSupply_InletValve_Open_A2" AND "Tag_7";   // falling edge of "q_xSupply_InletValve_Open_A2"
   "Tag_7" := "q_xSupply_InletValve_Open_A2";
   IF #_w1 THEN "i_xSupply_InletValve_Open_A2" := FALSE; END_IF;
   #_w2 := NOT "q_xSupply_FeedValve_Open_A2" AND "Tag_8";   // falling edge of "q_xSupply_FeedValve_Open_A2"
   "Tag_8" := "q_xSupply_FeedValve_Open_A2";
   IF #_w2 THEN "i_xSupply_FeedValve_Open_A2" := FALSE; END_IF;
END_REGION

REGION Network 7: INTERLOCKED VALVE
   RUNG wire#powerrail
      Contact( "i_xButtonSolenoidValve_Start" )
      wire#w1
      I_Contact( "i_xButtonSolenoidValve_Stop" )
      I_Contact( "q_xMix_Motor_Start" )
      Contact( "i_xMix_Tank_EmptySensor" )
      Coil( "i_xDrain_SolenoidValve_Open" )
   END_RUNG
   RUNG wire#powerrail
      Contact( "i_xDrain_SolenoidValve_Open" )
   END_RUNG wire#w1
   // the same network as SCL:
   "i_xDrain_SolenoidValve_Open" := ("i_xButtonSolenoidValve_Start" OR "i_xDrain_SolenoidValve_Open") AND NOT "i_xButtonSolenoidValve_Stop" AND NOT "q_xMix_Motor_Start" AND "i_xMix_Tank_EmptySensor";
END_REGION
END_FUNCTION_BLOCK

// folder: 01 Equipment/Functions

FUNCTION_BLOCK "FB - Supply_A1"   // FB4, LAD
{ S7_Optimized_Access := 'TRUE' }
VERSION : 0.1
   VAR_INPUT
      i_xPump_Running : Bool;
      i_xPump_Ready : Bool;
      i_xInletValve_Open : Bool;
      i_xFeedValve_Open : Bool;
      i_xLevel_Tank_Full : Bool;
      i_xSupply_FlowSensor : Bool;
      i_rLevel_Tank : Int;
   END_VAR
   VAR_OUTPUT
      q_xStart_Pump : Bool;
      q_xStop_Pump : Bool;
      q_xOpen_InletValve : Bool;
      q_xOpen_FeedValve : Bool;
   END_VAR
   VAR_IN_OUT
      iq_stStateHandler : "UDT_Statehandler";
      iq_stSupply : "UDT_Supply";
      iq_stDrain : "UDT_Drain";
      iq_stMix : "UDT_Mix";
   END_VAR
   VAR
      _xCmd_Start_Pump_A1 : Bool;
      _xCmd_Stop_Pump_A1 : Bool;
      xCmd_Open_InletValve_A1 : Bool;
      xCmd_Open_FeedValve_A1 : Bool;
   END_VAR
   VAR_TEMP
      _tTimeET : Time;
   END_VAR
BEGIN

REGION Network 1: OUTPUT - Start Pump
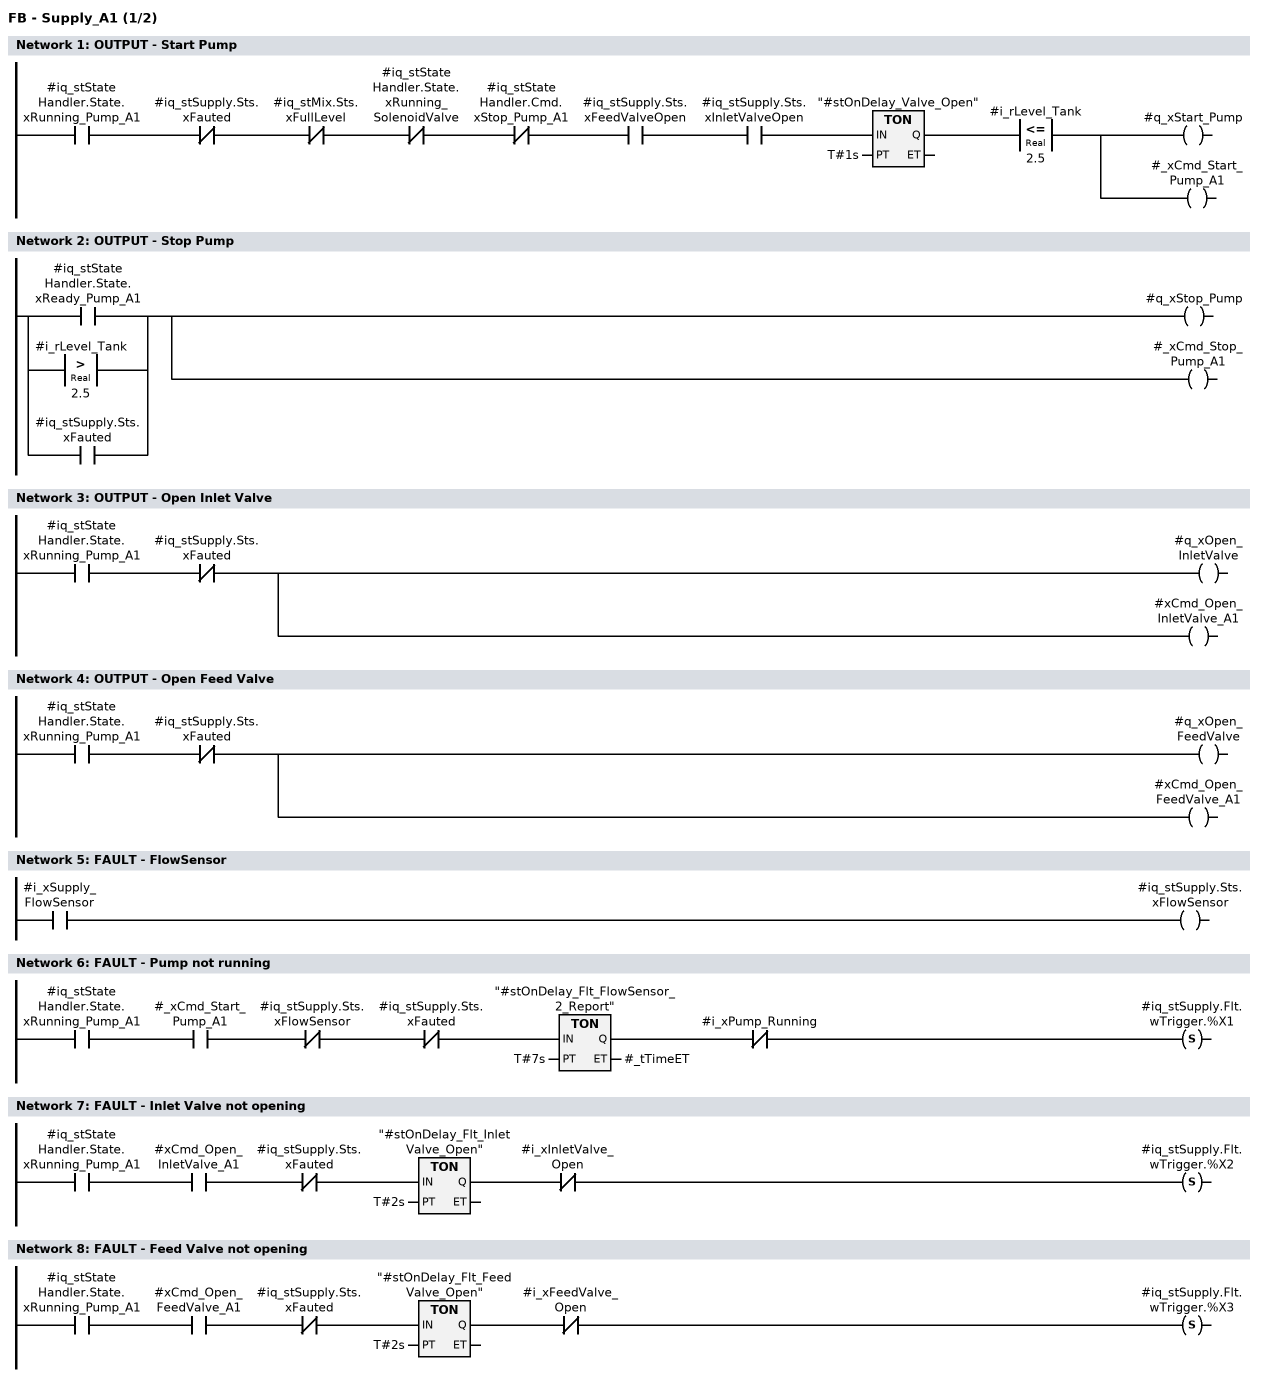
   "#stOnDelay_Valve_Open".TON(IN := #iq_stStateHandler.State.xRunning_Pump_A1 AND NOT #iq_stSupply.Sts.xFauted AND NOT #iq_stMix.Sts.xFullLevel AND NOT #iq_stStateHandler.State.xRunning_SolenoidValve AND NOT #iq_stStateHandler.Cmd.xStop_Pump_A1 AND #iq_stSupply.Sts.xFeedValveOpen AND #iq_stSupply.Sts.xInletValveOpen,
                           PT := T#1s);
   #q_xStart_Pump := "#stOnDelay_Valve_Open".Q AND (#i_rLevel_Tank <= 2.5);
   #_xCmd_Start_Pump_A1 := #q_xStart_Pump;
END_REGION

REGION Network 2: OUTPUT - Stop Pump
   RUNG wire#powerrail
      Contact( #iq_stStateHandler.State.xReady_Pump_A1 )
      wire#w1
      Coil( #q_xStop_Pump )
   END_RUNG
   RUNG wire#powerrail
      { S7_Templates := "SrcType := Real" } GT_Contact(in1 := #i_rLevel_Tank, in2 := 2.5)
   END_RUNG wire#w1
   RUNG wire#powerrail
      Contact( #iq_stSupply.Sts.xFauted )
   END_RUNG wire#w1
   RUNG wire#w1
      Coil( #_xCmd_Stop_Pump_A1 )
   END_RUNG
   // the same network as SCL:
   #q_xStop_Pump := #iq_stStateHandler.State.xReady_Pump_A1 OR (#i_rLevel_Tank > 2.5) OR #iq_stSupply.Sts.xFauted;
   #_xCmd_Stop_Pump_A1 := #q_xStop_Pump;
END_REGION

REGION Network 3: OUTPUT - Open Inlet Valve
   RUNG wire#powerrail
      Contact( #iq_stStateHandler.State.xRunning_Pump_A1 )
      I_Contact( #iq_stSupply.Sts.xFauted )
      wire#w1
      Coil( #q_xOpen_InletValve )
   END_RUNG
   RUNG wire#w1
      Coil( #xCmd_Open_InletValve_A1 )
   END_RUNG
   // the same network as SCL:
   #q_xOpen_InletValve := #iq_stStateHandler.State.xRunning_Pump_A1 AND NOT #iq_stSupply.Sts.xFauted;
   #xCmd_Open_InletValve_A1 := #q_xOpen_InletValve;
END_REGION

REGION Network 4: OUTPUT - Open Feed Valve
   RUNG wire#powerrail
      Contact( #iq_stStateHandler.State.xRunning_Pump_A1 )
      I_Contact( #iq_stSupply.Sts.xFauted )
      wire#w1
      Coil( #q_xOpen_FeedValve )
   END_RUNG
   RUNG wire#w1
      Coil( #xCmd_Open_FeedValve_A1 )
   END_RUNG
   // the same network as SCL:
   #q_xOpen_FeedValve := #iq_stStateHandler.State.xRunning_Pump_A1 AND NOT #iq_stSupply.Sts.xFauted;
   #xCmd_Open_FeedValve_A1 := #q_xOpen_FeedValve;
END_REGION

REGION Network 5: FAULT - FlowSensor
   RUNG wire#powerrail
      Contact( #i_xSupply_FlowSensor )
      Coil( #iq_stSupply.Sts.xFlowSensor )
   END_RUNG
   // the same network as SCL:
   #iq_stSupply.Sts.xFlowSensor := #i_xSupply_FlowSensor;
END_REGION

REGION Network 6: FAULT - Pump not running
   "#stOnDelay_Flt_FlowSensor_2_Report".TON(IN := #iq_stStateHandler.State.xRunning_Pump_A1 AND #_xCmd_Start_Pump_A1 AND NOT #iq_stSupply.Sts.xFlowSensor AND NOT #iq_stSupply.Sts.xFauted,
                           PT := T#7s,
                           ET => #_tTimeET);
   IF "#stOnDelay_Flt_FlowSensor_2_Report".Q AND NOT #i_xPump_Running THEN
       #iq_stSupply.Flt.wTrigger.%X1 := TRUE;
   END_IF;
END_REGION

REGION Network 7: FAULT - Inlet Valve not opening
   "#stOnDelay_Flt_Inlet Valve_Open".TON(IN := #iq_stStateHandler.State.xRunning_Pump_A1 AND #xCmd_Open_InletValve_A1 AND NOT #iq_stSupply.Sts.xFauted,
                           PT := T#2s);
   IF "#stOnDelay_Flt_Inlet Valve_Open".Q AND NOT #i_xInletValve_Open THEN
       #iq_stSupply.Flt.wTrigger.%X2 := TRUE;
   END_IF;
END_REGION

REGION Network 8: FAULT - Feed Valve not opening
   "#stOnDelay_Flt_Feed Valve_Open".TON(IN := #iq_stStateHandler.State.xRunning_Pump_A1 AND #xCmd_Open_FeedValve_A1 AND NOT #iq_stSupply.Sts.xFauted,
                           PT := T#2s);
   IF "#stOnDelay_Flt_Feed Valve_Open".Q AND NOT #i_xFeedValve_Open THEN
       #iq_stSupply.Flt.wTrigger.%X3 := TRUE;
   END_IF;
END_REGION

REGION Network 9: FAULT - Reset all fault
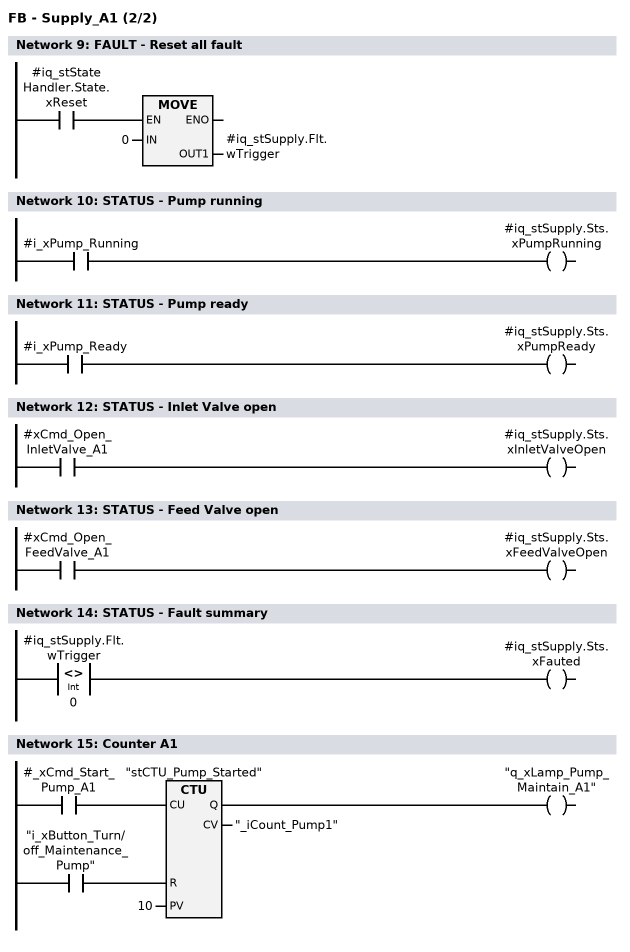
   RUNG wire#powerrail
      Contact( #iq_stStateHandler.State.xReset )
      Move(in := 0, out1 => #iq_stSupply.Flt.wTrigger)
   END_RUNG
   // the same network as SCL:
   IF #iq_stStateHandler.State.xReset THEN #iq_stSupply.Flt.wTrigger := 0; END_IF;
END_REGION

REGION Network 10: STATUS - Pump running
   RUNG wire#powerrail
      Contact( #i_xPump_Running )
      Coil( #iq_stSupply.Sts.xPumpRunning )
   END_RUNG
   // the same network as SCL:
   #iq_stSupply.Sts.xPumpRunning := #i_xPump_Running;
END_REGION

REGION Network 11: STATUS - Pump ready
   RUNG wire#powerrail
      Contact( #i_xPump_Ready )
      Coil( #iq_stSupply.Sts.xPumpReady )
   END_RUNG
   // the same network as SCL:
   #iq_stSupply.Sts.xPumpReady := #i_xPump_Ready;
END_REGION

REGION Network 12: STATUS - Inlet Valve open
   RUNG wire#powerrail
      Contact( #xCmd_Open_InletValve_A1 )
      Coil( #iq_stSupply.Sts.xInletValveOpen )
   END_RUNG
   // the same network as SCL:
   #iq_stSupply.Sts.xInletValveOpen := #xCmd_Open_InletValve_A1;
END_REGION

REGION Network 13: STATUS - Feed Valve open
   RUNG wire#powerrail
      Contact( #xCmd_Open_FeedValve_A1 )
      Coil( #iq_stSupply.Sts.xFeedValveOpen )
   END_RUNG
   // the same network as SCL:
   #iq_stSupply.Sts.xFeedValveOpen := #xCmd_Open_FeedValve_A1;
END_REGION

REGION Network 14: STATUS - Fault summary
   RUNG wire#powerrail
      { S7_Templates := "SrcType := Int" } NE_Contact(in1 := #iq_stSupply.Flt.wTrigger, in2 := 0)
      Coil( #iq_stSupply.Sts.xFauted )
   END_RUNG
   // the same network as SCL:
   #iq_stSupply.Sts.xFauted := #iq_stSupply.Flt.wTrigger <> 0;
END_REGION

REGION Network 15: Counter A1
   "stCTU_Pump_Started".CTU(CU := #_xCmd_Start_Pump_A1,
                           R := "i_xButton_Turn/off_Maintenance_Pump",
                           PV := 10,
                           CV => "_iCount_Pump1");
   "q_xLamp_Pump_Maintain_A1" := "stCTU_Pump_Started".Q;
END_REGION
END_FUNCTION_BLOCK

FUNCTION_BLOCK "FB - Agitator Motor"   // FB5, LAD
{ S7_Optimized_Access := 'TRUE' }
VERSION : 0.1
   VAR_INPUT
      i_xEmpty_Sensor : Bool := true;
      i_xFull_Sensor : Bool;
      i_rSpeed : Real := 1400.0;
      i_rLevel_Sensor : Real;
   END_VAR
   VAR_OUTPUT
      q_xStart_Motor : Bool;
      q_xVoltage_Supply : Real;
      q_xStop_Motor : Bool;
   END_VAR
   VAR_IN_OUT
      iq_stStateHandler : "UDT_Statehandler";
      iq_StDrain : "UDT_Drain";
      iq_stMix : "UDT_Mix";
   END_VAR
   VAR
      _xCmd_Open_Solenoid : Bool;
      _xCmd_Close_Solenoid : Bool;
      _xCmd_Start_Motor : Bool;
      _xCmd_Stop_Motor : Bool;
      _xMotor_Running : Bool;
   END_VAR
   VAR_TEMP
      _rSpeed1 : Real;
   END_VAR
BEGIN

REGION Network 1: INTERLOCKED
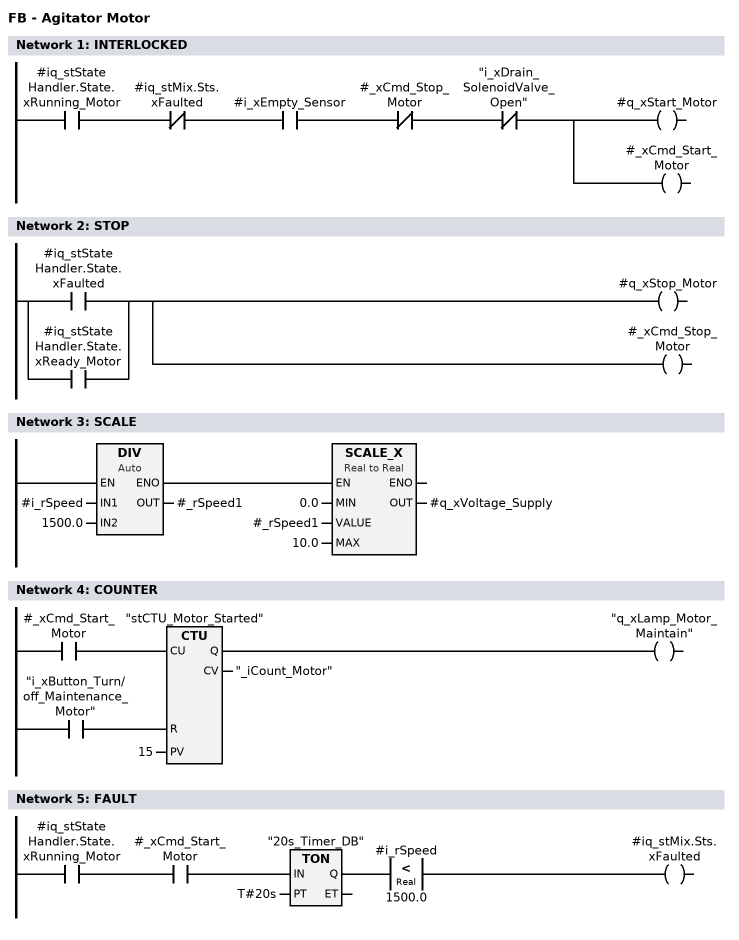
   RUNG wire#powerrail
      Contact( #iq_stStateHandler.State.xRunning_Motor )
      I_Contact( #iq_stMix.Sts.xFaulted )
      Contact( #i_xEmpty_Sensor )
      I_Contact( #_xCmd_Stop_Motor )
      I_Contact( "i_xDrain_SolenoidValve_Open" )
      wire#w1
      Coil( #q_xStart_Motor )
   END_RUNG
   RUNG wire#w1
      Coil( #_xCmd_Start_Motor )
   END_RUNG
   // the same network as SCL:
   #q_xStart_Motor := #iq_stStateHandler.State.xRunning_Motor AND NOT #iq_stMix.Sts.xFaulted AND #i_xEmpty_Sensor AND NOT #_xCmd_Stop_Motor AND NOT "i_xDrain_SolenoidValve_Open";
   #_xCmd_Start_Motor := #q_xStart_Motor;
END_REGION

REGION Network 2: STOP
   RUNG wire#powerrail
      Contact( #iq_stStateHandler.State.xFaulted )
      wire#w1
      Coil( #q_xStop_Motor )
   END_RUNG
   RUNG wire#powerrail
      Contact( #iq_stStateHandler.State.xReady_Motor )
   END_RUNG wire#w1
   RUNG wire#w1
      Coil( #_xCmd_Stop_Motor )
   END_RUNG
   // the same network as SCL:
   #q_xStop_Motor := #iq_stStateHandler.State.xFaulted OR #iq_stStateHandler.State.xReady_Motor;
   #_xCmd_Stop_Motor := #q_xStop_Motor;
END_REGION

REGION Network 3: SCALE
   RUNG wire#powerrail
      Div(in1 := #i_rSpeed, in2 := 1500.0, out => #_rSpeed1)
      { S7_Templates := "[SrcType := Real, DestType := Real]" } Scale(min := 0.0, value := #_rSpeed1, max := 10.0, out => #q_xVoltage_Supply)
   END_RUNG
   // the same network as SCL:
   #_rSpeed1 := #i_rSpeed / 1500.0;
   #q_xVoltage_Supply := SCALE_X(MIN := 0.0, VALUE := #_rSpeed1, MAX := 10.0);
END_REGION

REGION Network 4: COUNTER
   "stCTU_Motor_Started".CTU(CU := #_xCmd_Start_Motor,
                           R := "i_xButton_Turn/off_Maintenance_Motor",
                           PV := 15,
                           CV => "_iCount_Motor");
   "q_xLamp_Motor_Maintain" := "stCTU_Motor_Started".Q;
END_REGION

REGION Network 5: FAULT
   "20s_Timer_DB".TON(IN := #iq_stStateHandler.State.xRunning_Motor AND #_xCmd_Start_Motor, PT := T#20s);
   #iq_stMix.Sts.xFaulted := "20s_Timer_DB".Q AND (#i_rSpeed < 1500.0);
END_REGION
END_FUNCTION_BLOCK

FUNCTION_BLOCK "FB - Drain Valve"   // FB6, LAD
{ S7_Optimized_Access := 'TRUE' }
VERSION : 0.1
   VAR_INPUT
      i_xSolenoid_Opening : Bool;
      i_xSolenoid_Closed : Bool;
   END_VAR
   VAR_OUTPUT
      q_xOpen_Solenoid : Bool;
      q_xClose_Solenoid : Bool;
   END_VAR
   VAR_IN_OUT
      iq_stStateHandler : "UDT_Statehandler";
      iq_StDrain : "UDT_Drain";
      iq_stMix : "UDT_Mix";
   END_VAR
   VAR
      _xCmd_Open_Solenoid : Bool;
      _xCmd_Close_Solenoid : Bool;
   END_VAR
BEGIN

REGION Network 1: OUT- Open Drain Solenoid
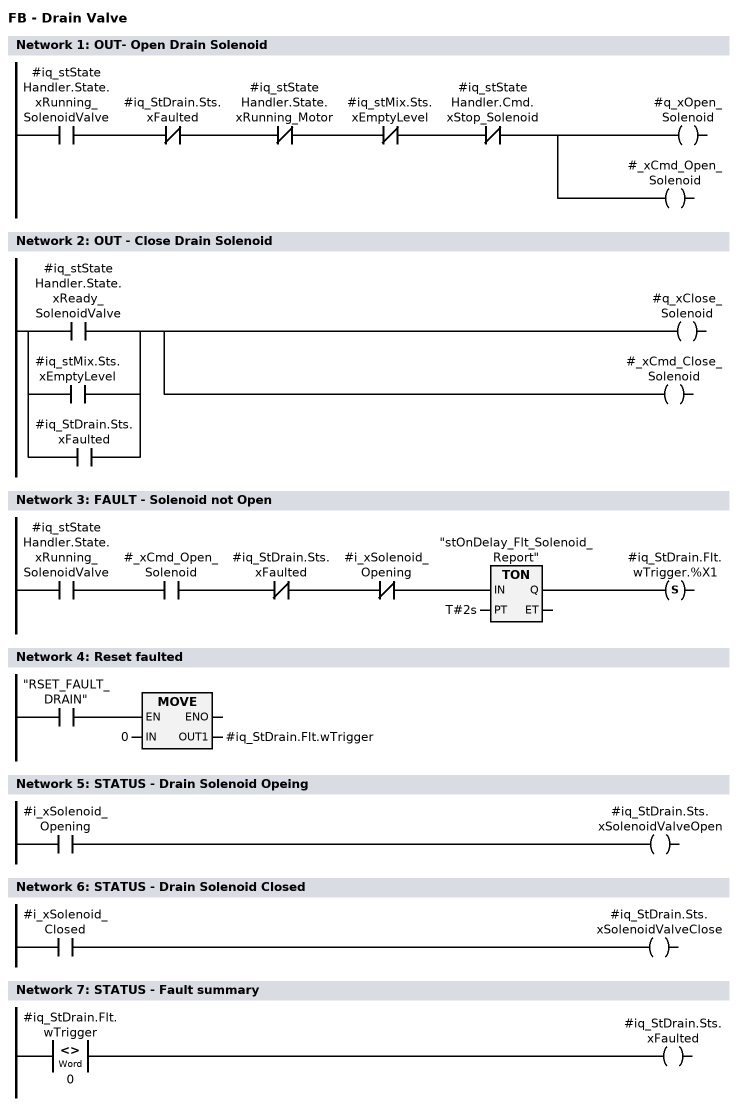
   RUNG wire#powerrail
      Contact( #iq_stStateHandler.State.xRunning_SolenoidValve )
      I_Contact( #iq_StDrain.Sts.xFaulted )
      I_Contact( #iq_stStateHandler.State.xRunning_Motor )
      I_Contact( #iq_stMix.Sts.xEmptyLevel )
      I_Contact( #iq_stStateHandler.Cmd.xStop_Solenoid )
      wire#w1
      Coil( #q_xOpen_Solenoid )
   END_RUNG
   RUNG wire#w1
      Coil( #_xCmd_Open_Solenoid )
   END_RUNG
   // the same network as SCL:
   #q_xOpen_Solenoid := #iq_stStateHandler.State.xRunning_SolenoidValve AND NOT #iq_StDrain.Sts.xFaulted AND NOT #iq_stStateHandler.State.xRunning_Motor AND NOT #iq_stMix.Sts.xEmptyLevel AND NOT #iq_stStateHandler.Cmd.xStop_Solenoid;
   #_xCmd_Open_Solenoid := #q_xOpen_Solenoid;
END_REGION

REGION Network 2: OUT - Close Drain Solenoid
   RUNG wire#powerrail
      Contact( #iq_stStateHandler.State.xReady_SolenoidValve )
      wire#w1
      Coil( #q_xClose_Solenoid )
   END_RUNG
   RUNG wire#powerrail
      Contact( #iq_stMix.Sts.xEmptyLevel )
   END_RUNG wire#w1
   RUNG wire#powerrail
      Contact( #iq_StDrain.Sts.xFaulted )
   END_RUNG wire#w1
   RUNG wire#w1
      Coil( #_xCmd_Close_Solenoid )
   END_RUNG
   // the same network as SCL:
   #q_xClose_Solenoid := #iq_stStateHandler.State.xReady_SolenoidValve OR #iq_stMix.Sts.xEmptyLevel OR #iq_StDrain.Sts.xFaulted;
   #_xCmd_Close_Solenoid := #q_xClose_Solenoid;
END_REGION

REGION Network 3: FAULT - Solenoid not Open
   "stOnDelay_Flt_Solenoid_Report".TON(IN := #iq_stStateHandler.State.xRunning_SolenoidValve AND #_xCmd_Open_Solenoid AND NOT #iq_StDrain.Sts.xFaulted AND NOT #i_xSolenoid_Opening,
                           PT := T#2s);
   IF "stOnDelay_Flt_Solenoid_Report".Q THEN #iq_StDrain.Flt.wTrigger.%X1 := TRUE; END_IF;
END_REGION

REGION Network 4: Reset faulted
   RUNG wire#powerrail
      Contact( "RSET_FAULT_DRAIN" )
      Move(in := 0, out1 => #iq_StDrain.Flt.wTrigger)
   END_RUNG
   // the same network as SCL:
   IF "RSET_FAULT_DRAIN" THEN #iq_StDrain.Flt.wTrigger := 0; END_IF;
END_REGION

REGION Network 5: STATUS - Drain Solenoid Opeing
   RUNG wire#powerrail
      Contact( #i_xSolenoid_Opening )
      Coil( #iq_StDrain.Sts.xSolenoidValveOpen )
   END_RUNG
   // the same network as SCL:
   #iq_StDrain.Sts.xSolenoidValveOpen := #i_xSolenoid_Opening;
END_REGION

REGION Network 6: STATUS - Drain Solenoid Closed
   RUNG wire#powerrail
      Contact( #i_xSolenoid_Closed )
      Coil( #iq_StDrain.Sts.xSolenoidValveClose )
   END_RUNG
   // the same network as SCL:
   #iq_StDrain.Sts.xSolenoidValveClose := #i_xSolenoid_Closed;
END_REGION

REGION Network 7: STATUS - Fault summary
   RUNG wire#powerrail
      { S7_Templates := "SrcType := Word" } NE_Contact(in1 := #iq_StDrain.Flt.wTrigger, in2 := 0)
      Coil( #iq_StDrain.Sts.xFaulted )
   END_RUNG
   // the same network as SCL:
   #iq_StDrain.Sts.xFaulted := #iq_StDrain.Flt.wTrigger <> 0;
END_REGION
END_FUNCTION_BLOCK

FUNCTION_BLOCK "FB - Supply_A2"   // FB7, LAD
{ S7_Optimized_Access := 'TRUE' }
VERSION : 0.1
   VAR_INPUT
      i_xPump_Running : Bool;
      i_xPump_Ready : Bool;
      i_xInletValve_Open : Bool;
      i_xFeedValve_Open : Bool;
      i_xLevel_Tank_Full : Bool;
      i_xSupply_FlowSensor : Bool;
   END_VAR
   VAR_OUTPUT
      q_xStart_Pump : Bool;
      q_xStop_Pump : Bool;
      q_xOpen_InletValve : Bool;
      q_xOpen_FeedValve : Bool;
   END_VAR
   VAR_IN_OUT
      iq_stStateHandler : "UDT_Statehandler";
      iq_stSupply : "UDT_Supply";
      iq_stDrain : "UDT_Drain";
      iq_stMix : "UDT_Mix";
   END_VAR
   VAR
      _xCmd_Start_Pump_A2 : Bool;
      _xCmd_Stop_Pump_A2 : Bool;
      xCmd_Open_InletValve_A2 : Bool;
      xCmd_Open_FeedValve_A2 : Bool;
   END_VAR
BEGIN

REGION Network 1: OUTPUT - Start Pump
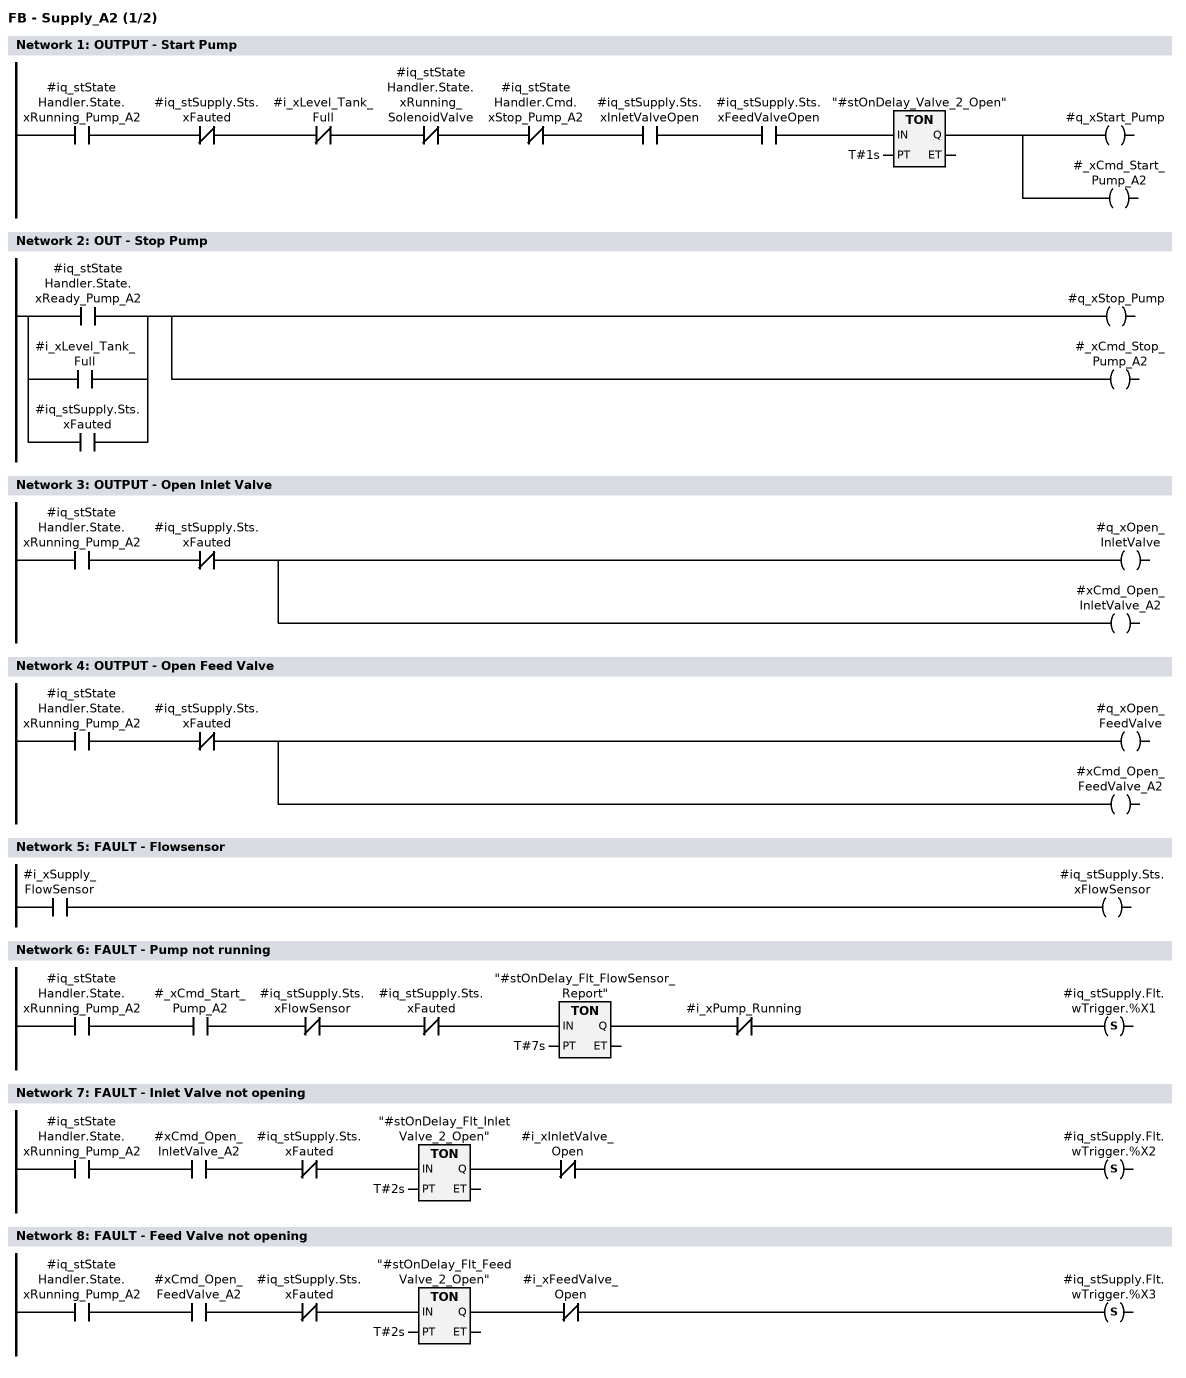
   "#stOnDelay_Valve_2_Open".TON(IN := #iq_stStateHandler.State.xRunning_Pump_A2 AND NOT #iq_stSupply.Sts.xFauted AND NOT #i_xLevel_Tank_Full AND NOT #iq_stStateHandler.State.xRunning_SolenoidValve AND NOT #iq_stStateHandler.Cmd.xStop_Pump_A2 AND #iq_stSupply.Sts.xInletValveOpen AND #iq_stSupply.Sts.xFeedValveOpen,
                           PT := T#1s);
   #q_xStart_Pump := "#stOnDelay_Valve_2_Open".Q;
   #_xCmd_Start_Pump_A2 := "#stOnDelay_Valve_2_Open".Q;
END_REGION

REGION Network 2: OUT - Stop Pump
   RUNG wire#powerrail
      Contact( #iq_stStateHandler.State.xReady_Pump_A2 )
      wire#w1
      Coil( #q_xStop_Pump )
   END_RUNG
   RUNG wire#powerrail
      Contact( #i_xLevel_Tank_Full )
   END_RUNG wire#w1
   RUNG wire#powerrail
      Contact( #iq_stSupply.Sts.xFauted )
   END_RUNG wire#w1
   RUNG wire#w1
      Coil( #_xCmd_Stop_Pump_A2 )
   END_RUNG
   // the same network as SCL:
   #q_xStop_Pump := #iq_stStateHandler.State.xReady_Pump_A2 OR #i_xLevel_Tank_Full OR #iq_stSupply.Sts.xFauted;
   #_xCmd_Stop_Pump_A2 := #q_xStop_Pump;
END_REGION

REGION Network 3: OUTPUT - Open Inlet Valve
   RUNG wire#powerrail
      Contact( #iq_stStateHandler.State.xRunning_Pump_A2 )
      I_Contact( #iq_stSupply.Sts.xFauted )
      wire#w1
      Coil( #q_xOpen_InletValve )
   END_RUNG
   RUNG wire#w1
      Coil( #xCmd_Open_InletValve_A2 )
   END_RUNG
   // the same network as SCL:
   #q_xOpen_InletValve := #iq_stStateHandler.State.xRunning_Pump_A2 AND NOT #iq_stSupply.Sts.xFauted;
   #xCmd_Open_InletValve_A2 := #q_xOpen_InletValve;
END_REGION

REGION Network 4: OUTPUT - Open Feed Valve
   RUNG wire#powerrail
      Contact( #iq_stStateHandler.State.xRunning_Pump_A2 )
      I_Contact( #iq_stSupply.Sts.xFauted )
      wire#w1
      Coil( #q_xOpen_FeedValve )
   END_RUNG
   RUNG wire#w1
      Coil( #xCmd_Open_FeedValve_A2 )
   END_RUNG
   // the same network as SCL:
   #q_xOpen_FeedValve := #iq_stStateHandler.State.xRunning_Pump_A2 AND NOT #iq_stSupply.Sts.xFauted;
   #xCmd_Open_FeedValve_A2 := #q_xOpen_FeedValve;
END_REGION

REGION Network 5: FAULT - Flowsensor
   RUNG wire#powerrail
      Contact( #i_xSupply_FlowSensor )
      Coil( #iq_stSupply.Sts.xFlowSensor )
   END_RUNG
   // the same network as SCL:
   #iq_stSupply.Sts.xFlowSensor := #i_xSupply_FlowSensor;
END_REGION

REGION Network 6: FAULT - Pump not running
   "#stOnDelay_Flt_FlowSensor_Report".TON(IN := #iq_stStateHandler.State.xRunning_Pump_A2 AND #_xCmd_Start_Pump_A2 AND NOT #iq_stSupply.Sts.xFlowSensor AND NOT #iq_stSupply.Sts.xFauted,
                           PT := T#7s);
   IF "#stOnDelay_Flt_FlowSensor_Report".Q AND NOT #i_xPump_Running THEN
       #iq_stSupply.Flt.wTrigger.%X1 := TRUE;
   END_IF;
END_REGION

REGION Network 7: FAULT - Inlet Valve not opening
   "#stOnDelay_Flt_Inlet Valve_2_Open".TON(IN := #iq_stStateHandler.State.xRunning_Pump_A2 AND #xCmd_Open_InletValve_A2 AND NOT #iq_stSupply.Sts.xFauted,
                           PT := T#2s);
   IF "#stOnDelay_Flt_Inlet Valve_2_Open".Q AND NOT #i_xInletValve_Open THEN
       #iq_stSupply.Flt.wTrigger.%X2 := TRUE;
   END_IF;
END_REGION

REGION Network 8: FAULT - Feed Valve not opening
   "#stOnDelay_Flt_Feed Valve_2_Open".TON(IN := #iq_stStateHandler.State.xRunning_Pump_A2 AND #xCmd_Open_FeedValve_A2 AND NOT #iq_stSupply.Sts.xFauted,
                           PT := T#2s);
   IF "#stOnDelay_Flt_Feed Valve_2_Open".Q AND NOT #i_xFeedValve_Open THEN
       #iq_stSupply.Flt.wTrigger.%X3 := TRUE;
   END_IF;
END_REGION

REGION Network 9: FAULT - Reset all fault
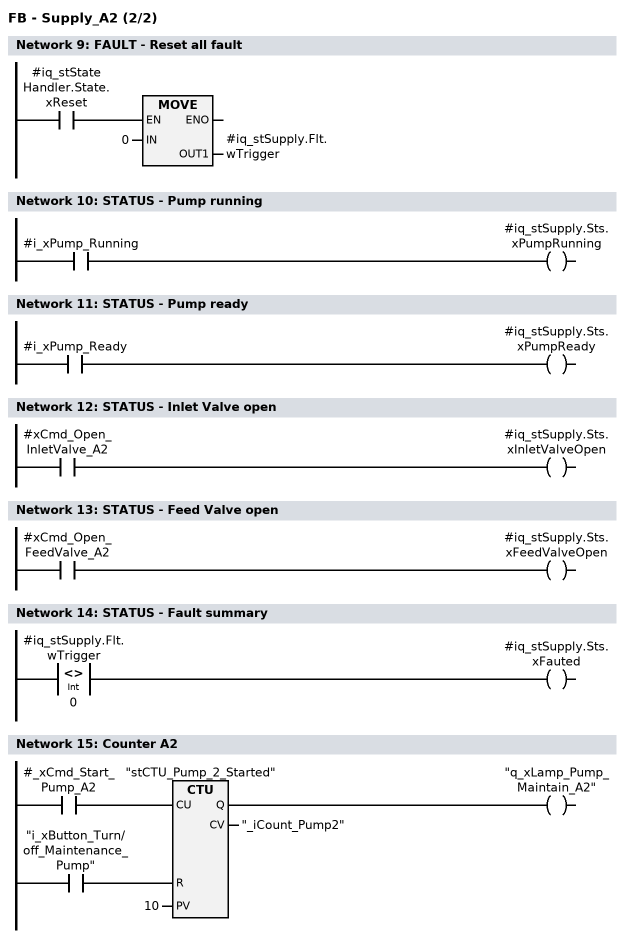
   RUNG wire#powerrail
      Contact( #iq_stStateHandler.State.xReset )
      Move(in := 0, out1 => #iq_stSupply.Flt.wTrigger)
   END_RUNG
   // the same network as SCL:
   IF #iq_stStateHandler.State.xReset THEN #iq_stSupply.Flt.wTrigger := 0; END_IF;
END_REGION

REGION Network 10: STATUS - Pump running
   RUNG wire#powerrail
      Contact( #i_xPump_Running )
      Coil( #iq_stSupply.Sts.xPumpRunning )
   END_RUNG
   // the same network as SCL:
   #iq_stSupply.Sts.xPumpRunning := #i_xPump_Running;
END_REGION

REGION Network 11: STATUS - Pump ready
   RUNG wire#powerrail
      Contact( #i_xPump_Ready )
      Coil( #iq_stSupply.Sts.xPumpReady )
   END_RUNG
   // the same network as SCL:
   #iq_stSupply.Sts.xPumpReady := #i_xPump_Ready;
END_REGION

REGION Network 12: STATUS - Inlet Valve open
   RUNG wire#powerrail
      Contact( #xCmd_Open_InletValve_A2 )
      Coil( #iq_stSupply.Sts.xInletValveOpen )
   END_RUNG
   // the same network as SCL:
   #iq_stSupply.Sts.xInletValveOpen := #xCmd_Open_InletValve_A2;
END_REGION

REGION Network 13: STATUS - Feed Valve open
   RUNG wire#powerrail
      Contact( #xCmd_Open_FeedValve_A2 )
      Coil( #iq_stSupply.Sts.xFeedValveOpen )
   END_RUNG
   // the same network as SCL:
   #iq_stSupply.Sts.xFeedValveOpen := #xCmd_Open_FeedValve_A2;
END_REGION

REGION Network 14: STATUS - Fault summary
   RUNG wire#powerrail
      { S7_Templates := "SrcType := Int" } NE_Contact(in1 := #iq_stSupply.Flt.wTrigger, in2 := 0)
      Coil( #iq_stSupply.Sts.xFauted )
   END_RUNG
   // the same network as SCL:
   #iq_stSupply.Sts.xFauted := #iq_stSupply.Flt.wTrigger <> 0;
END_REGION

REGION Network 15: Counter A2
   "stCTU_Pump_2_Started".CTU(CU := #_xCmd_Start_Pump_A2,
                           R := "i_xButton_Turn/off_Maintenance_Pump",
                           PV := 10,
                           CV => "_iCount_Pump2");
   "q_xLamp_Pump_Maintain_A2" := "stCTU_Pump_2_Started".Q;
END_REGION
END_FUNCTION_BLOCK

FUNCTION_BLOCK "FB - Motor's Speed"   // FB8, SCL
{ S7_Optimized_Access := 'TRUE' }
VERSION : 0.1
   VAR_INPUT
      Speed_Max : Real := 1500.0;
      tau : Real := 1.0;
      Ts : Real := 1.0;
      Power : Real := 1.0;
      Speed_1 : Real;
   END_VAR
   VAR_OUTPUT
      Speed : Real;
   END_VAR
   VAR
      Power_1 : Real;
   END_VAR
   VAR_TEMP
      "A" : Real;
      "B" : Real;
   END_VAR
BEGIN
   #A := EXP(- #Ts / #tau);
   #B := #Speed_Max * (1 - #A);
   #Speed := #A * #Speed_1 + #B * #Power_1;
   #Power_1 := #Power;
END_FUNCTION_BLOCK

FUNCTION_BLOCK "FB- Water's Level"   // FB9, SCL
{ S7_Optimized_Access := 'TRUE' }
VERSION : 0.1
   VAR_INPUT
      i_rQ : Real;
      i_rK : Real;
      i_rA : Real;
      i_iT : Int;
      rH1 : Real;
   END_VAR
   VAR_OUTPUT
      q_rH : Real;
      q_HLimit : Bool;
   END_VAR
   VAR
      rQ1 : Real;
   END_VAR
BEGIN
   #q_rH := #rH1 + (#rQ1 - #i_rK * SQRT(#rH1)) * #i_iT / #i_rA;
   #rQ1 := #i_rQ;

   IF #q_rH > 5.0 THEN
       #q_HLimit := 1;

   END_IF;
END_FUNCTION_BLOCK

ORGANIZATION_BLOCK "Cyclic interrupt"   // OB30, LAD, CyclicInterrupt
{ S7_Optimized_Access := 'TRUE' }
VERSION : 0.1
   VAR_INPUT
      Initial_Call : Bool;   // Initial call of this OB
      Event_Count : Int;   // Events discarded
   END_VAR
BEGIN

REGION Network 1
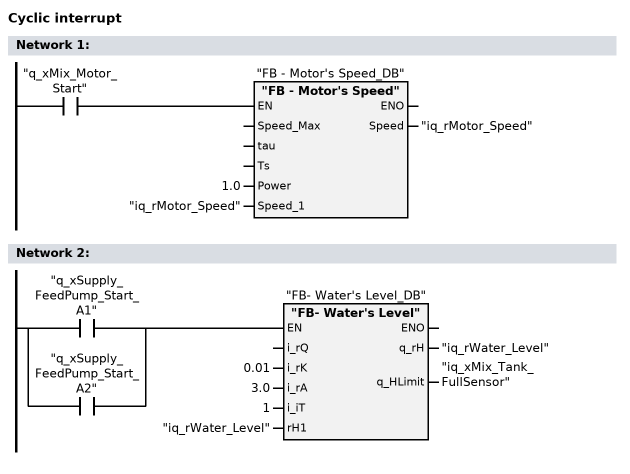
   RUNG wire#powerrail
      Contact( "q_xMix_Motor_Start" )
      "FB - Motor's Speed_DB"(Speed_Max :=, tau :=, Ts :=, Power := 1.0, Speed_1 := "iq_rMotor_Speed", Speed => "iq_rMotor_Speed")
   END_RUNG
   // the same network as SCL:
   IF "q_xMix_Motor_Start" THEN
       "FB - Motor's Speed_DB"(Power := 1.0, Speed_1 := "iq_rMotor_Speed", Speed => "iq_rMotor_Speed");   // "FB - Motor's Speed"
   END_IF;
END_REGION

REGION Network 2
   RUNG wire#powerrail
      Contact( "q_xSupply_FeedPump_Start_A1" )
      wire#w1
      "FB- Water's Level_DB"(i_rQ :=, i_rK := 0.01, i_rA := 3.0, i_iT := 1, rH1 := "iq_rWater_Level", q_rH => "iq_rWater_Level", q_HLimit => "iq_xMix_Tank_FullSensor")
   END_RUNG
   RUNG wire#powerrail
      Contact( "q_xSupply_FeedPump_Start_A2" )
   END_RUNG wire#w1
   // the same network as SCL:
   IF "q_xSupply_FeedPump_Start_A1" OR "q_xSupply_FeedPump_Start_A2" THEN
       "FB- Water's Level_DB"(i_rK := 0.01,   // "FB- Water's Level"
                              i_rA := 3.0,
                              i_iT := 1,
                              rH1 := "iq_rWater_Level",
                              q_rH => "iq_rWater_Level",
                              q_HLimit => "iq_xMix_Tank_FullSensor");
   END_IF;
END_REGION
END_ORGANIZATION_BLOCK

(* ===== HMI "HMI_RT_1" =====
system functions are stored by id; their names below are inferred from use
connection "HMI_Connection_1": ETHERNET, SMART_S7_1200_OMS
connection "HMI_Connection_2": ETHERNET, SMART_S7_1200_OMS
connection "HMI_Connection_3": ETHERNET, SMART_S7_1200_OMS

HMI tags "Default tag table"
   "Tag_ScreenNumber" : UInt, internal
   "q_xDisp_Tank_Level" : Real = PLC q_xDisp_Tank_Level AT %QD60, 1 s
   "iq_rWater_Level" : Real = PLC iq_rWater_Level AT %MD7, 1 s
   "iq_rMotor_Speed" : Real = PLC iq_rMotor_Speed AT %MD1, 1 s
   "i_xButtonMotor_Start" : Bool = PLC i_xButtonMotor_Start AT %I30.0, 1 s
   "i_xButtonMotor_Stop" : Bool = PLC i_xButtonMotor_Stop AT %I30.1, 1 s
   "i_xButtonFeedPump_Start_A1" : Bool = PLC i_xButtonFeedPump_Start_A1 AT %I30.3, 1 s
   "i_xButtonFeedPump_Stop_A1" : Bool = PLC i_xButtonFeedPump_Stop_A1 AT %I30.4, 1 s
   "i_xButtonFeedPump_Start_A2" : Bool = PLC i_xButtonFeedPump_Start_A2 AT %I30.5, 1 s
   "i_xButtonFeedPump_Stop_A2" : Bool = PLC i_xButtonFeedPump_Stop_A2 AT %I30.6, 1 s
   "i_xButtonSolenoidValve_Start" : Bool = PLC i_xButtonSolenoidValve_Start AT %I31.0, 1 s
   "i_xButtonSolenoidValve_Stop" : Bool = PLC i_xButtonSolenoidValve_Stop AT %I31.1, 1 s
   "i_xButton_Reset" : Bool = PLC i_xButton_Reset AT %I30.2, 1 s
   "i_xButton_Turn/off_Maintenance_Motor" : Bool = PLC "i_xButton_Turn/off_Maintenance_Motor" AT %I31.2, 1 s
   "i_xButton_Turn/off_Maintenance_Pump" : Bool = PLC "i_xButton_Turn/off_Maintenance_Pump" AT %I31.3, 1 s
   "_iCount_Motor" : Int = PLC _iCount_Motor AT %MW130, 1 s
   "_iCount_Pump1" : Int = PLC _iCount_Pump1 AT %MW115, 1 s
   "_iCount_Pump2" : Int = PLC _iCount_Pump2 AT %MW118, 1 s
   "q_xLamp_Motor_Stop" : Bool = PLC q_xLamp_Motor_Stop AT %Q4.7, 1 s
   "q_xLamp_Pump_Stop_A1" : Bool = PLC q_xLamp_Pump_Stop_A1 AT %Q4.3, 1 s
   "q_xLamp_Motor_Start" : Bool = PLC q_xLamp_Motor_Start AT %Q4.6, 1 s
   "q_xLamp_Pump_Start_A1" : Bool = PLC q_xLamp_Pump_Start_A1 AT %Q4.2, 1 s
   "q_xLamp_Pump_Start_A2" : Bool = PLC q_xLamp_Pump_Start_A2 AT %Q4.4, 1 s
   "q_xLamp_Pump_Stop_A2" : Bool = PLC q_xLamp_Pump_Stop_A2 AT %Q4.5, 1 s
   "q_xLamp_Fault" : Bool = PLC q_xLamp_Fault AT %Q120.1, 1 s

Template "Template_1" 800x480
   Button "Exit" at 714,429 size 71x50; TextOff 'Exit'; PictureOff "ExitRuntime_KTP700_Basic_PN_TR"; PictureOn "ExitRuntime_KTP700_Basic_PN_TR"
      on Release: StopRuntime(0)
   Button "Template_Button" at 614,429 size 71x50; TextOff 'Text'
   Button "Template_Button_1" at 514,429 size 71x50; TextOff 'Text'
   Button "Template_Button_2" at 414,429 size 71x50; TextOff 'Text'
   Button "Template_Button_3" at 314,429 size 71x50; TextOff 'Text'
   Button "Template_Button_4" at 214,429 size 71x50; TextOff 'Text'
   Button "Alarms" at 114,429 size 71x50; TextOff 'Alarms'; PictureOff "AlarmDisplay_KTP700_Basic_PN_TR"; PictureOn "AlarmDisplay_KTP700_Basic_PN_TR"
      on Release: function_ef3f5d25("Alarm window_Unacknowledged", -1)
   Button "Start screen" at 14,429 size 71x50; TextOff 'Start screen'; PictureOff "NavigateHome_KTP700_Basic_PN_TR"; PictureOn "NavigateHome_KTP700_Basic_PN_TR"
      on Release: ActivateScreen("Root screen", 0)
   SymbolicIOField "Symbolic_IO_Field_Screen" at 93,9 size 600x33; TextOff '0'; TextOn '1'; TextList "TextList_ScreenNames"
      ProcessValue <- "Tag_ScreenNumber"
      on Change: ActivateScreenByNumber("Tag_ScreenNumber", 0)
   DateTimeField "HmiScreenItemData" at 695,25 size 105x25
   DateTimeField "HmiScreenItemData_1" at 695,0 size 105x25
   GraphicView "Logo" at 0,0 size 91x51; Picture "Logo of HMI_1"

screen "Root screen" 800x480, template "Template_1"
   on GenerateScreen: SetTag("Tag_ScreenNumber", 1)
   Bar "Bar_1" at 433,211 size 173x212; MinimumValue 0; MaximumValue 7
      ProcessValue <- "iq_rWater_Level"
   IOField "I/O field_1" at 463,87 size 121x32; FormatPattern s999999999.999
      ProcessValue <- "iq_rMotor_Speed"
   Button "Button_2" at 43,114 size 124x48; TextOff 'Start Pump 1'
      on Release: ResetBit("i_xButtonFeedPump_Start_A1")
      on Press: SetBit("i_xButtonFeedPump_Start_A1")
   Button "Button_3" at 43,172 size 124x48; TextOff 'Start Pump 2'
      on Press: SetBit("i_xButtonFeedPump_Start_A2")
      on Release: ResetBit("i_xButtonFeedPump_Start_A2")
   Button "Button_4" at 186,59 size 124x48; TextOff 'Stop Motor'
      on Press: SetBit("i_xButtonMotor_Stop")
      on Release: ResetBit("i_xButtonMotor_Stop")
   Button "Button_5" at 186,114 size 124x48; TextOff 'Stop Pump 1'
      on Press: SetBit("i_xButtonFeedPump_Stop_A1")
      on Release: ResetBit("i_xButtonFeedPump_Stop_A1")
   Button "Button_6" at 183,172 size 124x48; TextOff 'Stop Pump 2'
      on Press: SetBit("i_xButtonFeedPump_Stop_A2")
      on Release: ResetBit("i_xButtonFeedPump_Stop_A2")
   Button "Button_7" at 43,238 size 181x52; TextOff 'Start Solenoid Valve'
      on Press: SetBit("i_xButtonSolenoidValve_Start")
      on Release: ResetBit("i_xButtonSolenoidValve_Start")
   Button "Button_8" at 44,302 size 180x49; TextOff 'Stop Solenoid Valve'
      on Press: SetBit("i_xButtonSolenoidValve_Stop")
      on Release: ResetBit("i_xButtonSolenoidValve_Stop")
   Button "Button_9" at 44,59 size 124x48; TextOff 'Start Motor'
      on Release: ResetBit("i_xButtonMotor_Start")
      on Press: SetBit("i_xButtonMotor_Start")
   Button "Button_10" at 43,361 size 124x48; TextOff 'Reset'
      on Release: ResetBit("i_xButton_Reset")
      on Press: SetBit("i_xButton_Reset")
   IOField "I/O field_2" at 476,161 size 96x32; FormatPattern s999999999.999
      ProcessValue <- "iq_rWater_Level"
   Button "Button_11" at 641,301 size 133x49; TextOff 'Maintain Motor'
      on Release: ResetBit("i_xButton_Turn/off_Maintenance_Motor")
      on Press: SetBit("i_xButton_Turn/off_Maintenance_Motor")
   Button "Button_12" at 641,361 size 133x50; TextOff 'Maintain Pump'
      on Release: ResetBit("i_xButton_Turn/off_Maintenance_Pump")
      on Press: SetBit("i_xButton_Turn/off_Maintenance_Pump")
   TextField "Text field_1" at 496,56 size 55x23; Text 'Speed'
   TextField "Text field_2" at 500,126 size 48x23; Text 'Level'
   IOField "I/O field_3" at 692,139 size 96x32; FormatPattern s99999
      ProcessValue <- "_iCount_Motor"
   IOField "I/O field_4" at 692,247 size 96x32; FormatPattern s99999
      ProcessValue <- "_iCount_Pump2"
   IOField "I/O field_5" at 692,193 size 96x32; FormatPattern s99999
      ProcessValue <- "_iCount_Pump1"
   TextField "Text field_3" at 624,144 size 53x23; Text 'Motor'
   TextField "Text field_4" at 620,193 size 61x23; Text 'Pump1'
   TextField "Text field_5" at 620,247 size 61x23; Text 'Pump2'
   TextField "Text field_6" at 706,101 size 53x23; Text 'Count'
   Circle "Circle_1" at 330,123 size 38x38
      Appearance <- "q_xLamp_Pump_Start_A1"
   Circle "Circle_2" at 382,123 size 38x38
      Appearance <- "q_xLamp_Pump_Stop_A1"
   Circle "Circle_3" at 330,63 size 38x38
      Appearance <- "q_xLamp_Motor_Start"
   Circle "Circle_4" at 330,182 size 38x38
      Appearance <- "q_xLamp_Pump_Start_A2"
   Circle "Circle_5" at 382,182 size 38x38
      Appearance <- "q_xLamp_Pump_Stop_A2"
   Circle "Circle_6" at 382,64 size 38x38
      Appearance <- "q_xLamp_Motor_Stop"
   Circle "Circle_7" at 298,290 size 84x84
      Appearance <- "q_xLamp_Fault"
*)